	axisSlave:=             arrAxis[AxiseNo.VirAxisName.VirMain], 
	axisMaster:=          arrAxis[AxiseNo.VirAxisName.VirDriver]    , 
	bCreatTableDone=> , 
	bCreatTableError=> , 
	bError=>  );

fbCreatCamVirGMDriver.bCreatTableDone;
fbCreatCamVirGMDriver.bCreatTableError;
fbCreatCamVirGMDriver.bError;

(***********隔膜摆臂凸轮表**************)
fbCreatCamGMDanserMove(
	bCreatTable:=                     fbCreatCamGMDanserMove.bCreatTable, 
	Reset:=                                stSysState.bReset  , 
	iTable_L:=                            TableNo.M_GMDanserMove_L , //3
	iTable_R:=                           TableNo.M_GMDanserMove_R, //6
    fMoveLength:=                     fMaxPos-fMinPos , 
    fMasterKeyPos:=                   250  , //180
	axisSlave:=                           arrAxis[AxiseNo.VirAxisName.VirMain]  , 
	axisMaster:=                        arrAxis[AxiseNo.AxisName.SEPTATLine] , 
	bCreatTableDone=> , 
	bCreatTableError=> , 
	bError=>  );

fbCreatCamGMDanserMove.bCreatTableDone;
fbCreatCamGMDanserMove.bCreatTableError;
fbCreatCamGMDanserMove.bError;


(***********************************************************隔膜缓存凸轮表创建V2***20240229**************************************************************************)
(*******极片缓存电机*********)
fbCreatCamGMBuffer2_L(
	Reset:=                              stSysState.bReset  , 
	bCreatTable:=                   fbCreatCamGMBuffer2_L.bCreatTable, 
	iTable:=                            TableNo.M_GMBuffer2_L , 
	iTableGMVirDriver:=          TableNo.M_GMWind2_L  , 
	iTableGMStackCalculate:=  TableNo.M_GMLengthCalculate2_L , 
	iTableGMStackMove:=       TableNo.M_GMDanserMove_L , 
	fMaxPos:=                           fMaxPos, 
	fMinPos:=                            fMinPos , 
    iCcwSel :=                          1 , 
	arrGMCalculateTableData:= arrDeltaGMLength2_L , 

	axisSlave:=                     arrAxis[AxiseNo.AxisName.SEPTATCache], 
	axisMaster:=                  arrAxis[AxiseNo.VirAxisName.VirMain] , 
	bCreatTableDone=> , 
	bCreatTableError=> , 
	bError=>  );
fbCreatCamGMBuffer2_L.bCreatTableDone;
fbCreatCamGMBuffer2_L.bCreatTableError;
fbCreatCamGMBuffer2_L.bError;


(*******极片缓存电机*********)
fbCreatCamGMBuffer2_R(
	Reset:=                              stSysState.bReset  , 
	bCreatTable:=                    fbCreatCamGMBuffer2_R.bCreatTable, 
	iTable:=                             TableNo.M_GMBuffer2_R , 
	iTableGMVirDriver:=           TableNo.M_GMWind2_R  , 
	iTableGMStackCalculate:=   TableNo.M_GMLengthCalculate2_R , 
	iTableGMStackMove:=         TableNo.M_GMDanserMove_R , 
    iCcwSel :=                           2 , 
   	fMaxPos:=                           fMaxPos, 
	fMinPos:=                            fMinPos , 
	arrGMCalculateTableData:= arrDeltaGMLength2_R , 

	axisSlave:=                     arrAxis[AxiseNo.AxisName.SEPTATCache], 
	axisMaster:=                  arrAxis[AxiseNo.VirAxisName.VirMain] , 
	bCreatTableDone=> , 
	bCreatTableError=> , 
	bError=>  );
fbCreatCamGMBuffer2_R.bCreatTableDone;
fbCreatCamGMBuffer2_R.bCreatTableError;
fbCreatCamGMBuffer2_R.bError;


(***********隔膜放卷虚轴*凸轮表**************)
fbCreatCamVirGMDriver2(
	bCreatTable:=         fbCreatCamVirGMDriver2.bCreatTable , 
	Reset:=                  stSysState.bReset, 
	iTable_L:=               TableNo.M_GMWind2_L , 
	iTable_R:=               TableNo.M_GMWind2_R , 

	fGMLength_L:=		arrDeltaGMLength2_L[3600,1], 
	fGMLength_R:=	arrDeltaGMLength2_R[3600,1],  

	axisSlave:=            arrAxis[AxiseNo.VirAxisName.VirDriver], 
	axisMaster:=        arrAxis[AxiseNo.VirAxisName.VirMain]       , 
	bCreatTableDone=> , 
	bCreatTableError=> , 
	bError=>  );

fbCreatCamVirGMDriver2.bCreatTableDone;
fbCreatCamVirGMDriver2.bCreatTableError;
fbCreatCamVirGMDriver2.bError;


tGMCreateCamTON(IN:= , PT:=T#0.5S , Q=> , ET=> );
IF Mach_Control.U.DT_iMode=3 OR Mach_Control.U.DT_iMode=0 THEN//在手动状态下
			//从触据屏创建隔膜缓存凸轮
			rGMCreateCam_TRIG(CLK:=Mach_Control.DT_b.CreateCamStart2 , Q=> );
			IF rGMCreateCam_TRIG.Q THEN
				tGMCreateCamTON.IN:=FALSE;
				GMCreatCamStep0:=10;
				Mach_Control.DT_b.Error[1]:=FALSE;
			END_IF
END_IF			
			//隔膜缓存凸轮创建 
			CASE GMCreatCamStep0 OF
						10:
								IF NOT 	tGMCreateCamTON.Q THEN
										fbCreatCamVirGMDriver.bCreatTable:=FALSE;//放卷凸轮创建
										fbCreatCamGMDanserMove.bCreatTable:=FALSE;//	隔膜平移凸轮创建
										fbCreatCamGMBuffer_L.bCreatTable:=FALSE;//缓存左凸轮生成
										fbCreatCamGMBuffer_R.bCreatTable:=FALSE;//缓存右轮生成
										Mach_Control.DT_b.CreateCamDone2:=FALSE;
										tGMCreateCamTON.IN:=TRUE;
								ELSE
										tGMCreateCamTON.IN:=FALSE;
										GMCreatCamStep0:=11;
								END_IF
			
						11:
							IF  NOT DT_Cam_ton[3].Q THEN
								arrAxisCtrl[AxiseNo.AxisName.SEPTAunwinding].Cmd.bStop:=TRUE;
								arrAxisCtrl[AxiseNo.AxisName.SEPTATCache].Cmd.bStop:=TRUE;
								arrAxisCtrl[AxiseNo.AxisName.SEPTATLine].Cmd.bStop:=TRUE;
								DT_Cam_ton[3].IN:=TRUE;
							ELSE
								DT_Cam_ton[3].IN:=FALSE;
								GMCreatCamStep0:=12;
								arrAxisCtrl[AxiseNo.AxisName.SEPTAunwinding].Cmd.bStop:=FALSE;
								arrAxisCtrl[AxiseNo.AxisName.SEPTATCache].Cmd.bStop:=FALSE;
								arrAxisCtrl[AxiseNo.AxisName.SEPTATLine].Cmd.bStop:=FALSE;
							END_IF
					
						12:
							IF  NOT DT_Cam_ton[4].Q THEN
								arrAxisCtrl[AxiseNo.AxisName.SEPTAunwinding].Cmd.bReset:=TRUE;	
								arrAxisCtrl[AxiseNo.AxisName.SEPTATCache].Cmd.bReset:=TRUE;
								arrAxisCtrl[AxiseNo.AxisName.SEPTATLine].Cmd.bReset:=TRUE;		
								DT_Cam_ton[4].IN:=TRUE;
							 ELSE
								 DT_Cam_ton[4].IN:=FALSE;
								 GMCreatCamStep0:=13;
								arrAxisCtrl[AxiseNo.AxisName.SEPTAunwinding].Cmd.bReset:=FALSE;	
								arrAxisCtrl[AxiseNo.AxisName.SEPTATCache].Cmd.bReset:=FALSE;
								arrAxisCtrl[AxiseNo.AxisName.SEPTATLine].Cmd.bReset:=FALSE;		
							 END_IF
								
						13:
							arrAxisCtrl[AxiseNo.AxisName.SEPTAunwinding].Cmd.bEnable:=TRUE;
							arrAxisCtrl[AxiseNo.AxisName.SEPTATCache].Cmd.bEnable:=TRUE;
							arrAxisCtrl[AxiseNo.AxisName.SEPTATLine].Cmd.bEnable:=TRUE;
							IF arrAxisCtrl[AxiseNo.AxisName.SEPTAunwinding].Status.Enabled AND arrAxisCtrl[AxiseNo.AxisName.SEPTATCache].Status.Enabled AND
								arrAxisCtrl[AxiseNo.AxisName.SEPTATLine].Status.Enabled THEN
								 GMCreatCamStep0:=20;
							END_IF				
								
							
						20://隔膜变化长度度算
								iSetp1:=10;
								iSetp2:=10;
								Mach_Control.DT_b.CreateCamDone2:=FALSE;
								GMCreatCamStep0:=30;
						30://等待隔膜变化长度计算完成
								IF iSetp1=666 AND iSetp2=666 THEN
									GMCreatCamStep0:=40;
								END_IF
						40://创建放卷凸轮、隔膜平移凸轮
								fbCreatCamVirGMDriver.bCreatTable:=TRUE;//放卷凸轮创建
								 fbCreatCamGMDanserMove.bCreatTable:=TRUE;//	隔膜平移凸轮创建
								 fbCreatCamVirGMDriver2.bCreatTable:=TRUE;//放卷凸轮创建
								 
								GMCreatCamStep0:=50;	
						50://等待凸轮创建完成
								IF fbCreatCamVirGMDriver.bCreatTableDone AND fbCreatCamGMDanserMove.bCreatTableDone AND  fbCreatCamVirGMDriver2.bCreatTableDone  THEN
									GMCreatCamStep0:=60;	
								ELSE
										IF fbCreatCamVirGMDriver.bCreatTableError OR fbCreatCamGMDanserMove.bCreatTableError OR   fbCreatCamVirGMDriver2.bCreatTableError  THEN
												Mach_Control.DT_b.Error[1]:=TRUE;//隔膜缓存凸轮创建失败
												GMCreatCamStep0:=9999;		
										END_IF					
								END_IF
						60://创建隔膜缓存凸轮
							fbCreatCamGMBuffer_L.bCreatTable:=TRUE;//缓存左凸轮生成
							fbCreatCamGMBuffer_R.bCreatTable:=TRUE;//缓存右轮生成
							fbCreatCamGMBuffer2_L.bCreatTable:=TRUE;//缓存左凸轮生成
							fbCreatCamGMBuffer2_R.bCreatTable:=TRUE;//缓存右轮生成		
							
							 //fbCamInVirGM.bCreatTable:=TRUE;//隔膜虚轴凸轮生成
							GMCreatCamStep0:=70;	
						70://等待凸轮创建完成
							IF fbCreatCamGMBuffer_L.bCreatTableDone AND fbCreatCamGMBuffer_R.bCreatTableDone (*  AND fbCamInVirGM.bCreatTableDone *)    AND 
                                fbCreatCamGMBuffer2_L.bCreatTableDone AND  fbCreatCamGMBuffer2_R.bCreatTableDone THEN
								Mach_Control.DT_b.CreateCamDone2:=TRUE;//隔膜缓存凸轮创建完成
								GMCreatCamStep0:=6666;	
							ELSE
									IF fbCreatCamGMBuffer_L.bCreatTableError OR fbCreatCamGMBuffer_R.bCreatTableError  OR 
                                         fbCreatCamGMBuffer2_L.bCreatTableError AND  fbCreatCamGMBuffer2_R.bCreatTableError THEN
										Mach_Control.DT_b.Error[1]:=TRUE;//隔膜缓存凸轮创建失败
										GMCreatCamStep0:=9999;	
									END_IF
							END_IF
			END_CASE
(************************************************************凸轮耦合*****************************************************************************)
//隔膜放卷凸轮
fbCamInVirGMDriver(  
	Reset:=                      stSysState.bReset  , 
	bCamInExecute:=       fbCamInVirGMDriver.bCamInExecute, 
	iTable1:=                   TableNo.M_GMWind_L  , //从左到右，正极到负极
	iTable2:=                  TableNo.M_GMWind_R  , //从右到左，负极到正极
	iTableSel:=                fbCamInVirGMDriver.iTableSel , //凸轮表号选择
	ParCamIn:= , 
 	axisMaster:=            arrAxis[AxiseNo.VirAxisName.VirMain], 
	axisSlave:=               arrAxis[AxiseNo.VirAxisName.VirDriver]    , 
	bError=> , 
	bReady=> , 
	bInSync=> );

Mach_Control.DT_b.Error[16]:=fbCamInVirGMDriver.bError;
fbCamInVirGMDriver.bReady;
fbCamInVirGMDriver.bInSync;


//隔膜平移凸轮
IF  fbCamInGMDanserMove.iTableSel=2 THEN
     fbCamInGMDanserMove.ParCamIn.SlaveOffset:=-(fMaxPos-fMinPos);
ELSE
    fbCamInGMDanserMove.ParCamIn.SlaveOffset:=0;
END_IF

fbCamInGMDanserMove(
	Reset:=                      stSysState.bReset  , 
	bCamInExecute:=       fbCamInGMDanserMove.bCamInExecute, 
	iTable1:=                   TableNo.M_GMDanserMove_L  , 
	iTable2:=                   TableNo.M_GMDanserMove_R  , 
	iTableSel:=                fbCamInGMDanserMove.iTableSel , 
	ParCamIn:= , 
  	axisMaster:=            arrAxis[AxiseNo.VirAxisName.VirMain] , //VirMain
	axisSlave:=               arrAxis[AxiseNo.AxisName.SEPTATLine] , 
	bError=> , 
	bReady=> , 
	bInSync=> );

Mach_Control.DT_b.Error[17]:=fbCamInGMDanserMove.bError;
fbCamInGMDanserMove.bReady;
fbCamInGMDanserMove.bInSync;

//隔膜缓存凸轮
fbCamInGMBuffer.ParCamIn.MasterScaling:=0.1;
fbCamInGMBuffer(
	Reset:=                      stSysState.bReset  , 
	bCamInExecute:=       fbCamInGMBuffer.bCamInExecute, 
	iTable1:=                   TableNo.M_GMBuffer_L  , 
	iTable2:=                   TableNo.M_GMBuffer_R  , 
	iTableSel:=                fbCamInGMBuffer.iTableSel , 
	ParCamIn:= , 
  	axisMaster:=           arrAxis[AxiseNo.VirAxisName.VirMain] , 
	axisSlave:=               arrAxis[AxiseNo.AxisName.SEPTATCache] , 
	bError=> , 
	bReady=> , 
	bInSync=> );

Mach_Control.DT_b.Error[18]:=fbCamInGMBuffer.bError;
fbCamInGMBuffer.bReady;
fbCamInGMBuffer.bInSync;



(************************************************************凸轮耦合V2*****************************************************************************)
//隔膜放卷凸轮
fbCamInVirGMDriver2(  
	Reset:=                      stSysState.bReset  , 
	bCamInExecute:=       fbCamInVirGMDriver2.bCamInExecute, 
	iTable1:=                   TableNo.M_GMWind2_L  , //从左到右，正极到负极
	iTable2:=                  TableNo.M_GMWind2_R  , //从右到左，负极到正极
	iTableSel:=                fbCamInVirGMDriver2.iTableSel , //凸轮表号选择
	ParCamIn:= , 
 	axisMaster:=            arrAxis[AxiseNo.VirAxisName.VirMain], 
	axisSlave:=               arrAxis[AxiseNo.VirAxisName.VirDriver]    , 
	bError=> , 
	bReady=> , 
	bInSync=> );

fbCamInVirGMDriver2.bError;
fbCamInVirGMDriver2.bReady;
fbCamInVirGMDriver2.bInSync;


//隔膜缓存凸轮
fbCamInGMBuffer2.ParCamIn.MasterScaling:=0.1;
fbCamInGMBuffer2(
	Reset:=                      stSysState.bReset  , 
	bCamInExecute:=       fbCamInGMBuffer2.bCamInExecute, 
	iTable1:=                   TableNo.M_GMBuffer2_L  , 
	iTable2:=                   TableNo.M_GMBuffer2_R  , 
	iTableSel:=                fbCamInGMBuffer2.iTableSel , 
	ParCamIn:= , 
  	axisMaster:=           arrAxis[AxiseNo.VirAxisName.VirMain] , 
	axisSlave:=               arrAxis[AxiseNo.AxisName.SEPTATCache] , 
	bError=> , 
	bReady=> , 
	bInSync=> );

fbCamInGMBuffer2.bError;
fbCamInGMBuffer2.bReady;
fbCamInGMBuffer2.bInSync;












(*

(***********************************************************隔膜缓存凸轮表创建*****************************************************************************)
(*******极片缓存电机*********)
fbCreatCamGMBuffer_L.iKeyPosTemp:=20;
fbCreatCamGMBuffer_L(
	Reset:=                              stSysState.bReset  , 
	bCreatTable:=                   fbCreatCamGMBuffer_L.bCreatTable, 
	iTable:=                            TableNo.M_GMBuffer_L , //10
	iTableGMVirDriver:=          TableNo.M_GMWind_L  , //1
	iTableGMStackCalculate:=  TableNo.M_GMLengthCalculate_L , //2
	iTableGMStackMove:=       TableNo.M_GMDanserMove_L , //3
	fMaxPos:=                           fMaxPos, 
	fMinPos:=                            fMinPos , 
    iCcwSel :=                          1 , 
	arrGMCalculateTableData:= arrDeltaGMLength_L , 

	axisSlave:=                     arrAxis[AxiseNo.VirAxisName.VirMain], 
	axisMaster:=                  arrAxis[AxiseNo.AxisName.SEPTATCache] , 
	bCreatTableDone=> , 
	bCreatTableError=> , 
	bError=>  );
fbCreatCamGMBuffer_L.bCreatTableDone;
fbCreatCamGMBuffer_L.bCreatTableError;
fbCreatCamGMBuffer_L.bError;


(*******极片缓存电机*********)
fbCreatCamGMBuffer_R.iKeyPosTemp:=20;
fbCreatCamGMBuffer_R(
	Reset:=                              stSysState.bReset  , 
	bCreatTable:=                    fbCreatCamGMBuffer_R.bCreatTable, 
	iTable:=                             TableNo.M_GMBuffer_R , //20
	iTableGMVirDriver:=           TableNo.M_GMWind_R  , //4
	iTableGMStackCalculate:=   TableNo.M_GMLengthCalculate_R , //5
	iTableGMStackMove:=         TableNo.M_GMDanserMove_R , //6
    iCcwSel :=                           2 , //2
   	fMaxPos:=                           fMaxPos, 
	fMinPos:=                            fMinPos , 
	arrGMCalculateTableData:= arrDeltaGMLength_R , 

	axisSlave:=                     arrAxis[AxiseNo.VirAxisName.VirMain], 
	axisMaster:=                  arrAxis[AxiseNo.AxisName.SEPTATCache] , 
	bCreatTableDone=> , 
	bCreatTableError=> , 
	bError=>  );
fbCreatCamGMBuffer_R.bCreatTableDone;
fbCreatCamGMBuffer_R.bCreatTableError;
fbCreatCamGMBuffer_R.bError;


(***********隔膜放卷虚轴*凸轮表**************)
fbCreatCamVirGMDriver(
	bCreatTable:=         fbCreatCamVirGMDriver.bCreatTable , 
	Reset:=                  stSysState.bReset, 
	iTable_L:=               TableNo.M_GMWind_L , //1
	iTable_R:=               TableNo.M_GMWind_R , //4

	fGMLength_L:=       arrDeltaGMLength_L[3600,1]+1.2 , 
	fGMLength_R:=       arrDeltaGMLength_R[3600,1]+1.2 , 

	axisSlave:=             arrAxis[AxiseNo.VirAxisName.VirMain], 
	axisMaster:=          arrAxis[AxiseNo.VirAxisName.VirDriver]    , 
	bCreatTableDone=> , 
	bCreatTableError=> , 
	bError=>  );

fbCreatCamVirGMDriver.bCreatTableDone;
fbCreatCamVirGMDriver.bCreatTableError;
fbCreatCamVirGMDriver.bError;
*)
END_ACTION

ACTION GMBufferLengthCalculate:
(**************************************************************************隔膜计算V2******************************************)


(**************************************************************************隔膜变化长度计算********************************************)
//隔膜垂直向下为隔膜摆臂的机械零点
//C1点坐标=当前坐标+隔膜辊半径
//fMaxPos=隔膜摆臂右目标位置+隔膜辊半径

(*
//C1活动范围   -188.05------164.05        从右到左 
(**********坐标自动计算**********)
Par.Mechaical.fGMRollDiameter:=24;
IF Par.Mechaical.fGM_X>0 AND Par.Mechaical.fGM_Y>0 THEN
	Par.Mechaical.y_B1:=Par.Mechaical.fGM_Y-Par.Mechaical.fGMRollDiameter/2;
	Par.Mechaical.y_C1:=Par.Mechaical.y_B1-72;
	//Par.Mechaical.y_A5:=Par.Mechaical.y_B1+333;
	Par.Mechaical.x_D2:=Par.Mechaical.fGM_X+52.5;
	Par.Mechaical.x_D1:=Par.Mechaical.x_D2-par.stDT_date.Width;
END_IF
IF Par.Mechaical.fGM_Z>0 THEN
	Par.Mechaical.y_A5:=Par.Mechaical.fGM_Z+Par.Mechaical.fGMRollDiameter/2;
END_IF
*)
       
arrAxisPar [AxiseNo.AxisName.SEPTATLine].arrTargetPoint[1];//左
arrAxisPar [AxiseNo.AxisName.SEPTATLine].arrTargetPoint[2];//右
Par.Mechaical.fGMRollDiameter;
CASE  iSetp1  OF   
10://计算相间距
    I10:=0;
	//fMaxPos:=arrAxisPar [AxiseNo.AxisName.SEPTATLine].arrTargetPoint[2]-arrAxisPar [AxiseNo.AxisName.SEPTATLine].arrTargetPoint[3] -Par.Mechaical.fGMRollDiameter/2;
	//fMinPos:=arrAxisPar [AxiseNo.AxisName.SEPTATLine].arrTargetPoint[1]-arrAxisPar [AxiseNo.AxisName.SEPTATLine].arrTargetPoint[3] -Par.Mechaical.fGMRollDiameter/2;	
	fMaxPos:=arrAxisPar [AxiseNo.AxisName.SEPTATLine].arrTargetPoint[2]-Par.Mechaical.fGMRollDiameter/2;
	fMinPos:=arrAxisPar [AxiseNo.AxisName.SEPTATLine].arrTargetPoint[1]-Par.Mechaical.fGMRollDiameter/2;
  // fMaxPos:=164.05;         //  =隔膜摆臂当前位置-r              隔膜摆臂中间为0位置
   //fMinPos:=-200;          //  =隔膜摆臂当前位置-r              隔膜摆臂中间为0位置          -188.55
    iNumberOfPoint:=3600;
    fInterval:=(fMaxPos-fMinPos)/ iNumberOfPoint ;


    fradii:= Par.Mechaical.fGMRollDiameter/2 ;
    fJumpPos:=-fradii;
    k_Comp:=fcompensationPos/(fMaxPos-fJumpPos) ;
	bMoveFowerdR:=FALSE;
    iSetp1:=20;

20:
   fTagatPos:=fMaxPos-I10*fInterval;
   bExecute:=TRUE;
   bExecute2:=TRUE;
    iSetp1:=30;
30:
   IF NOT  bExecute   AND  NOT bExecute2   THEN
        arrfTagatPos_R[I10]:=fTagatPos;
        arrDeltaGMLength_R[I10,0]:=I10;
 
       arrGMLengthDown_R[I10] :=fbGMLengthV1_R.fTotalLenght;
       arrGMLengthUp_R[I10] :=fbGMLengthV2_R.fTotalLenght   ;
		
       arrDeltaGMLength_R[0,1]:=0;
       IF I10>=1 THEN
         arrDeltaGMLength_R[I10,1]:=arrGMLengthDown_R[I10]+arrGMLengthUp_R[I10]-(arrGMLengthDown_R[0]+arrGMLengthUp_R[0] )        ;
      END_IF
          I10:=I10+1;
		IF I10>iNumberOfPoint THEN
			iSetp1:=100;  
		ELSE
			iSetp1:=20;  
		 END_IF
   END_IF

100:
       I10:=0;
	//fMaxPos:=arrAxisPar [AxiseNo.AxisName.SEPTATLine].arrTargetPoint[2]-arrAxisPar [AxiseNo.AxisName.SEPTATLine].arrTargetPoint[3] -Par.Mechaical.fGMRollDiameter/2;
	//fMinPos:=arrAxisPar [AxiseNo.AxisName.SEPTATLine].arrTargetPoint[1]-arrAxisPar [AxiseNo.AxisName.SEPTATLine].arrTargetPoint[3] -Par.Mechaical.fGMRollDiameter/2;	
	fMaxPos:=arrAxisPar [AxiseNo.AxisName.SEPTATLine].arrTargetPoint[2]-Par.Mechaical.fGMRollDiameter/2;
	fMinPos:=arrAxisPar [AxiseNo.AxisName.SEPTATLine].arrTargetPoint[1]-Par.Mechaical.fGMRollDiameter/2;
  // fMaxPos:=164.05;         //  =隔膜摆臂当前位置-r              隔膜摆臂中间为0位置
   //fMinPos:=-200;          //  =隔膜摆臂当前位置-r              隔膜摆臂中间为0位置          -188.55
    iNumberOfPoint:=3600;
    fInterval:=(fMaxPos-fMinPos)/ iNumberOfPoint ;


    fradii:= Par.Mechaical.fGMRollDiameter/2 ;
    fJumpPos:=-fradii;
    k_Comp:=fcompensationPos/(fMaxPos-fJumpPos) ;
   bMoveFowerdR:=TRUE;
    iSetp1:=120;

120:
     fTagatPos:=fMaxPos-I10*fInterval;
     bExecute:=TRUE;
     bExecute2:=TRUE;
      iSetp1:=130;

130:
	IF NOT  bExecute   AND  NOT bExecute2   THEN
			arrfTagatPos2_R[I10]:=fTagatPos;
			arrDeltaGMLength2_R[I10,0]:=I10;
			
			arrGMLengthDown2_R[I10] :=fbGMLengthV1_R.fTotalLenght;
			arrDeltaGMLength2_R[0,1]:=0;
			IF I10>=1 THEN
				arrDeltaGMLength2_R[I10,1]:=arrGMLengthDown2_R[I10]+arrGMLengthUp_R[I10]-(arrGMLengthDown2_R[0]+arrGMLengthUp_R[0] )        ;
			END_IF
			I10:=I10+1;
			IF I10>iNumberOfPoint THEN
				iSetp1:=666;  
			ELSE
				iSetp1:=120;  
			END_IF
		END_IF 
END_CASE



//C1活动范围   -188.05------164.05        从左到右   
CASE  iSetp2  OF   
10://计算相间距
    I12:=0;
	fMaxPos:=arrAxisPar [AxiseNo.AxisName.SEPTATLine].arrTargetPoint[2]-Par.Mechaical.fGMRollDiameter/2;
	fMinPos:=arrAxisPar [AxiseNo.AxisName.SEPTATLine].arrTargetPoint[1]-Par.Mechaical.fGMRollDiameter/2;
  // fMaxPos:=164.05;       
   // fMinPos:=-200;  
    iNumberOfPoint:=3600;
    fInterval2:=(fMaxPos-fMinPos)/ iNumberOfPoint ;
 
    fradii:= Par.Mechaical.fGMRollDiameter/2 ;
    fJumpPos:=-fradii;
    k_Comp:=fcompensationPos/(fMaxPos-fJumpPos) ;

     arrDeltaGMLengthAbs_L[0,0]:=0 ;
	 bMoveFowerdL:=FALSE;
    iSetp2:=20;

20:
   fTagatPos2:=fMinPos+I12*fInterval2;
   bExecute3:=TRUE;
   bExecute4:=TRUE;
    iSetp2:=30;

30:
   IF NOT  bExecute3   AND  NOT bExecute4   THEN
        arrfTagatPos_L[I12]:=fTagatPos2;
        arrDeltaGMLength_L[I12,0]:=I12;
        arrDeltaGMLengthAbs_L[I12,0]:=fTagatPos2-fMinPos ;

        arrGMLengthDown_L[I12] :=  fbGMLengthV1_L.fTotalLenght;  //下
         arrGMLengthUp_L[I12] :=fbGMLengthV2_L.fTotalLenght   ;  //上	
		
      arrDeltaGMLength_L[0,1]:=0;
       IF I12>=1 THEN
         arrDeltaGMLength_L[I12,1]:=arrDeltaGMLengthAbs_L[I12,1]:= arrGMLengthDown_L[I12]+arrGMLengthUp_L[I12]-(arrGMLengthDown_L[0]+arrGMLengthUp_L[0] )   ;
      END_IF
          I12:=I12+1;
		IF I12>iNumberOfPoint THEN
			iSetp2:=100;  
		ELSE
			iSetp2:=20;  
		 END_IF
   END_IF

100:
    I12:=0;
	fMaxPos:=arrAxisPar [AxiseNo.AxisName.SEPTATLine].arrTargetPoint[2]-Par.Mechaical.fGMRollDiameter/2;
	fMinPos:=arrAxisPar [AxiseNo.AxisName.SEPTATLine].arrTargetPoint[1]-Par.Mechaical.fGMRollDiameter/2;
  // fMaxPos:=164.05;       
   // fMinPos:=-200;  
    iNumberOfPoint:=3600;
    fInterval2:=(fMaxPos-fMinPos)/ iNumberOfPoint ;
 
    fradii:= Par.Mechaical.fGMRollDiameter/2 ;
    fJumpPos:=-fradii;
    k_Comp:=fcompensationPos/(fMaxPos-fJumpPos) ;

     arrDeltaGMLength2Abs_L[0,0]:=0 ;
	 bMoveFowerdL:=TRUE;
    iSetp2:=120;
	 
120:	 
	   fTagatPos2:=fMinPos+I12*fInterval2;
	   bExecute3:=TRUE;
	   bExecute4:=TRUE;
		iSetp2:=130;	 
130:	 
  IF NOT  bExecute3   AND  NOT bExecute4   THEN
        arrfTagatPos2_L[I12]:=fTagatPos2;
        arrDeltaGMLength2_L[I12,0]:=I12;
        arrDeltaGMLength2Abs_L[I12,0]:=fTagatPos2-fMinPos ;
		
        arrGMLengthDown2_L[I12] :=  fbGMLengthV1_L.fTotalLenght;  //下
       // arrGMLengthUp_L[I12] :=fbGMLengthV2_L.fTotalLenght   ;  //上	
      arrDeltaGMLength2_L[0,1]:=0;
       IF I12>=1 THEN
         arrDeltaGMLength2_L[I12,1]:=arrDeltaGMLength2Abs_L[I12,1]:= arrGMLengthDown2_L[I12]+arrGMLengthUp_L[I12]-(arrGMLengthDown2_L[0]+arrGMLengthUp_L[0] )  ;
      END_IF
          I12:=I12+1;
		IF I12>iNumberOfPoint THEN
			iSetp2:=666;  
		ELSE
			iSetp2:=120;  
		 END_IF

   END_IF	 
	
END_CASE


(***从右往左运动*)
fbGMLengthV1_R(
	bExecute:=           bExecute , 
     x_C1:=                  fTagatPos, 

    fradii:=                       Par.Mechaical.fGMRollDiameter/2 , 
    y_C1:=                       Par.Mechaical.y_C1    , 
    x_D1:=                      SEL(bMoveFowerdR,Par.Mechaical.x_D1,Par.Mechaical.x_D1)    , //
    x_D2:=                      SEL(bMoveFowerdR,Par.Mechaical.x_D2,Par.Mechaical.x_D1)  , //20221028  SJ
	fDegree=> , 
	fArcLength=> , 
	fLineLength=> , 
	fTotalLenght=> );
fbGMLengthV1_R.fArcLength;
fbGMLengthV1_R.fDegree;
fbGMLengthV1_R.fLineLength;
fbGMLengthV1_R.fTotalLenght;


(*
fbGMLengthV2_R(
	x_C1:=                           fTagatPos , 

   fradii:=                       Par.Mechaical.fGMRollDiameter/2 , 
    y_C1:=                       Par.Mechaical.y_C1    , 
    x_D1:=                       Par.Mechaical.x_D1   , 
    x_D2:=                       Par.Mechaical.x_D2  , 
    y_B1:=                       Par.Mechaical.y_B1   , 
    y_A5:=                       Par.Mechaical.y_A5   , 

	fDegree=> , 
	fArcLength=> , 
	fLineLength=> , 
	fTotalLenght=> , 
	bExecute:=                    bExecute2 );

fbGMLengthV2_R.fArcLength;
fbGMLengthV2_R.fDegree;
fbGMLengthV2_R.fLineLength;
fbGMLengthV2_R.fTotalLenght;
*)

fbGMLengthV2_R(
	x_C1:=                           fTagatPos , 

   fradii:=                       Par.Mechaical.fGMRollDiameter/2 , 
    y_C1:=                       Par.Mechaical.y_C1    , 
    x_D1:=                       Par.Mechaical.x_D1   , 
    x_D2:=                       Par.Mechaical.x_D2  , 
    y_B1:=                       Par.Mechaical.y_B1   , 
    y_A5:=                       Par.Mechaical.y_A5   , 

	fDegree=> , 
	fArcLength=> , 
	fLineLength=> , 
	fTotalLenght=> , 
	bExecute:=                    bExecute2 );

fbGMLengthV2_R.fArcLength;
fbGMLengthV2_R.fDegree;
fbGMLengthV2_R.fLineLength;
fbGMLengthV2_R.fTotalLenght;


(***从左往右运动*)
fbGMLengthV1_L(  //下
	bExecute:=             bExecute3 , 
     x_C1:=                  fTagatPos2, 

    fradii:=                       Par.Mechaical.fGMRollDiameter/2 , 
    y_C1:=                       Par.Mechaical.y_C1    , 
    x_D1:=                         SEL(bMoveFowerdL,Par.Mechaical.x_D1,Par.Mechaical.x_D2)  , // x_D1:=x_D2;//20221028SJ
    x_D2:=                       SEL(bMoveFowerdL,Par.Mechaical.x_D2,Par.Mechaical.x_D2)  , // x_D1:=x_D2;//20221028SJ

	fDegree=> , 
	fArcLength=> , 
	fLineLength=> , 
	fTotalLenght=> );
fbGMLengthV1_L.fArcLength;
fbGMLengthV1_L.fDegree;
fbGMLengthV1_L.fLineLength;
fbGMLengthV1_L.fTotalLenght;


(*
fbGMLengthV2_L( //上
	x_C1:=                        fTagatPos2 , 
    
    fradii:=                       Par.Mechaical.fGMRollDiameter/2 , 
    y_C1:=                       Par.Mechaical.y_C1    , 
    x_D1:=                       Par.Mechaical.x_D1   , 
    x_D2:=                       Par.Mechaical.x_D2  , 
    y_B1:=                       Par.Mechaical.y_B1   , 
    y_A5:=                       Par.Mechaical.y_A5   , 

	fDegree=> , 
	fArcLength=> , 
	fLineLength=> , 
	fTotalLenght=> , 
	bExecute:=                    bExecute4 );

fbGMLengthV2_L.fArcLength;
fbGMLengthV2_L.fDegree;
fbGMLengthV2_L.fLineLength;
fbGMLengthV2_L.fTotalLenght;
*)
fbGMLengthV2_L( //上
	x_C1:=                        fTagatPos2 , 
    
    fradii:=                       Par.Mechaical.fGMRollDiameter/2 , 
    y_C1:=                       Par.Mechaical.y_C1    , 
    x_D1:=                       Par.Mechaical.x_D1   , 
    x_D2:=                       Par.Mechaical.x_D2  , 
    y_B1:=                       Par.Mechaical.y_B1   , 
    y_A5:=                       Par.Mechaical.y_A5   , 

	fDegree=> , 
	fArcLength=> , 
	fLineLength=> , 
	fTotalLenght=> , 
	bExecute:=                    bExecute4 );

fbGMLengthV2_L.fArcLength;
fbGMLengthV2_L.fDegree;
fbGMLengthV2_L.fLineLength;
fbGMLengthV2_L.fTotalLenght;




fbReadCamSlavePos(
	Execute:=              fbReadCamSlavePos.Execute , 
	CamTableID:=        1, 
	MasterPosition:=    fbReadCamSlavePos.MasterPosition, 
	Done=> , 
	Busy=> , 
	Error=> , 
	ErrorID=> , 
	SlavePosition=> , 
	SlaveVelocity=> , 
	SlaveAcceleration=> );

fbReadCamSlavePos.Done;
fbReadCamSlavePos.Error;
fbReadCamSlavePos.SlavePosition;
END_ACTION

ACTION GMEmptyFold1:
//首层隔膜空叠自动步	iEmptyFoldStep[1]
DT_AlarmTon[5](IN:=  , PT:=T#300MS , Q=> , ET=> );
	
IF Mach_Control.U.DT_iMode=1 THEN//在自动状态下
CASE iEmptyFoldStep[1] OF
100:
   DT_AlarmTon[5].IN:=FALSE;
   IF NOT DP_SinStepe THEN
		IF NOT  Mach_Control.DT_b.DT_YDOpenwindow THEN
			CCD.Over.Start.iPliesNo:=UINT_TO_INT(Mach_Control.Ca_b.Ca_Quantited + Mach_Control.An_b.An_Quantited);
			CCD.Over.Finish.OverhandResult:=0;
			Mach_Control.DT_b.OverhandResult:=0;
			CCD.Over.Start.iPhotoDo:=3;
			Mach_Control.DT_b.CDD_OverStart:=TRUE;
			iEmptyFoldStep[1]:=200;
		ELSE
			iEmptyFoldStep[1]:=900;
		END_IF
    END_IF
200:
DT_AlarmTon[5].IN:=TRUE;
IF Mach_Control.DT_b.OverhandResult=1 THEN
	CellMemory[Mach_Control.DT_b.DT_Memory].Overhang_Result[CCD.Over.Start.iPliesNo]:=Mach_Control.DT_b.OverhandResult;
	iEmptyFoldStep[1]:=900;
ELSIF Mach_Control.DT_b.OverhandResult=5 THEN
	Mach_Control.DT_b.Error[63]:=TRUE;//首次对齐度拍照NG，请调节压刀间距
	iEmptyFoldStep[1]:=100;
ELSIF DT_AlarmTon[5].Q THEN
	Mach_Control.DT_b.Error[65]:=TRUE;//压刀间距测量结果返馈超时
	iEmptyFoldStep[1]:=100;
	DT_AlarmTon[5].IN :=FALSE;
END_IF



900://判断主轴是否停止、是否在初始位、是否有轴在耦合中
	bEmptyFoldMark[1]:=TRUE;//进入空叠流程
	IF NOT DP_SinStepe THEN
		bFirstFoldFinish[1]:=FALSE;//首层隔膜空叠完成
		IF arrAxisCtrl[AxiseNo.VirAxisName.VirMain].Status.NoMoving AND arrAxisCtrl[AxiseNo.VirAxisName.VirMain].Status.fSetPos=0 AND NOT DT_AxiseCoupling THEN
			DT_SingeMode();//单步选择	
			iEmptyFoldStep[1]:=1020;
		ELSE
			DT_SingeMode();//单步选择	
			DP_Step1:=100;//解除耦合，主轴回零
			iEmptyFoldStep[1]:=1010;
		END_IF
	END_IF
1010://判断主轴当前的当前位置是否为0
	IF DP_Step1=6666 AND arrAxisCtrl[AxiseNo.VirAxisName.VirMain].Status.NoMoving AND arrAxisCtrl[AxiseNo.VirAxisName.VirMain].Status.fSetPos=0 AND NOT DT_AxiseCoupling THEN
		DT_SingeMode();//单步选择
		iEmptyFoldStep[1]:=1020;						
	END_IF	

1020://判断NG气缸是否在安全位
	IF arrCyCtrl[arrCyNo.CylinderName.AnScrapbinCy].Status.ONState AND arrCyCtrl[arrCyNo.CylinderName.CaScrapbinUDCy].Status.OFFState AND
		arrCyCtrl[arrCyNo.CylinderName.CaScrapbinCy].Status.ONState AND arrCyCtrl[arrCyNo.CylinderName.PreDiaph].Status.OFFState AND 
		arrCyCtrl[arrCyNo.CylinderName.PoleHotCutterCy].Status.OFFState AND arrCyCtrl[arrCyNo.CylinderName.PoleTapeCy].Status.OFFState AND
		arrCyCtrl[arrCyNo.CylinderName.PoleTapeSplicerRCy].Status.ONState AND arrCyCtrl[arrCyNo.CylinderName.PoleTapeSplicerLCy].Status.ONState THEN
		iEmptyFoldStep[1]:=1050;		
	ELSE
		iEmptyFoldStep[1]:=1030;	
	END_IF
1030:
	IF NOT DP_SinStepe THEN
		arrCyCtrl[arrCyNo.CylinderName.AnScrapbinCy].Cmd.bON:=TRUE;
		arrCyCtrl[arrCyNo.CylinderName.PreDiaph].Cmd.bOFF:=TRUE;
		arrCyCtrl[arrCyNo.CylinderName.PoleHotCutterCy].Cmd.bOFF:=TRUE;
		arrCyCtrl[arrCyNo.CylinderName.PoleTapeCy].Cmd.bOFF:=TRUE;
		arrCyCtrl[arrCyNo.CylinderName.PoleTapeSplicerRCy].Cmd.bON:=TRUE;
		arrCyCtrl[arrCyNo.CylinderName.PoleTapeSplicerLCy].Cmd.bON:=TRUE;
		arrCyCtrl[arrCyNo.CylinderName.CaScrapbinCy].Cmd.bON:=TRUE;
		IF   arrCyCtrl[arrCyNo.CylinderName.AnScrapbinCy].Status.ONState AND  arrCyCtrl[arrCyNo.CylinderName.PreDiaph].Status.OFFState AND 
		arrCyCtrl[arrCyNo.CylinderName.PoleHotCutterCy].Status.OFFState AND arrCyCtrl[arrCyNo.CylinderName.PoleTapeCy].Status.OFFState AND
		arrCyCtrl[arrCyNo.CylinderName.PoleTapeSplicerRCy].Status.ONState AND arrCyCtrl[arrCyNo.CylinderName.PoleTapeSplicerLCy].Status.ONState
		AND arrCyCtrl[arrCyNo.CylinderName.CaScrapbinCy].Cmd.bON THEN
			DT_SingeMode();//单步选择	
			iEmptyFoldStep[1]:=1040;									
		END_IF
	END_IF	
1040:
	IF NOT DP_SinStepe THEN
		arrCyCtrl[arrCyNo.CylinderName.CaScrapbinUDCy].Cmd.bOFF:=TRUE;
		IF  arrCyCtrl[arrCyNo.CylinderName.CaScrapbinUDCy].Status.OFFState THEN
			DT_SingeMode();//单步选择	
			iEmptyFoldStep[1]:=1050;	
		END_IF		
	END_IF				
1050://	首层空叠隔膜
	IF Mach_Control.An_b.An_FirstFoldCnt<=Mach_Control.Ca_b.Ca_FirstFoldCnt THEN//先叠正极
		iEmptyFoldStep[1]:=1100;
	ELSIF Mach_Control.An_b.An_FirstFoldCnt>Mach_Control.Ca_b.Ca_FirstFoldCnt  THEN//先叠负极
		iEmptyFoldStep[1]:=1500;
	END_IF	
1100://判断叠台搬运机械手是否有片
	IF AN_CarryingPos1  THEN//正极搬运、叠片各轴在初始位	
		IF arrCyCtrl[arrCyNo.ElectValveName.AnDTCarryingVacuum].Io.DIOnSwitch AND  Mach_Control.An_b.An_DPCarryingFalg THEN//正极再取片位且叠台搬运有片,把当前片放到纠偏台
			iEmptyFoldStep[1]:=1150;
		ELSE
			iEmptyFoldStep[1]:=2000;	
		END_IF
	ELSE
		Mach_Control.DT_b.Error[8]:=TRUE;//叠正极片凸轮耦合时，正极片不在取片位
		//DP_Step0:=10001;
	END_IF	
	
1150://纠偏台回初始位
	//纠偏平台X1移动至初始位
	IF NOT DP_SinStepe THEN
		IF arrAxisCtrl[AxiseNo.AxisName.AndeviationX1].Status.Homed  AND arrAxisCtrl[AxiseNo.AxisName.AndeviationX1].Status.NoMoving AND NOT  arrAxisCtrl[AxiseNo.AxisName.AndeviationX1].Status.Error THEN
			IF arrAxisCtrl[AxiseNo.AxisName.AndeviationX1].Cmd.arrbRealPoint[1] THEN
				arrAxisCtrl[AxiseNo.AxisName.AndeviationX1].Cmd.iGoSetPos:=0;
			ELSE
				arrAxisCtrl[AxiseNo.AxisName.AndeviationX1].Cmd.iGoSetPos:=1;
			END_IF					
		END_IF
		//纠偏平台X2移动至初始位
		IF arrAxisCtrl[AxiseNo.AxisName.AndeviationX2].Status.Homed  AND arrAxisCtrl[AxiseNo.AxisName.AndeviationX2].Status.NoMoving AND NOT  arrAxisCtrl[AxiseNo.AxisName.AndeviationX2].Status.Error THEN
			IF arrAxisCtrl[AxiseNo.AxisName.AndeviationX2].Cmd.arrbRealPoint[1] THEN
				arrAxisCtrl[AxiseNo.AxisName.AndeviationX2].Cmd.iGoSetPos:=0;
			ELSE
				arrAxisCtrl[AxiseNo.AxisName.AndeviationX2].Cmd.iGoSetPos:=1;
			END_IF					
		END_IF
		//纠偏平台X2移动至初始位
		IF arrAxisCtrl[AxiseNo.AxisName.AndeviationY].Status.Homed  AND arrAxisCtrl[AxiseNo.AxisName.AndeviationY].Status.NoMoving AND NOT  arrAxisCtrl[AxiseNo.AxisName.AndeviationY].Status.Error THEN
			IF arrAxisCtrl[AxiseNo.AxisName.AndeviationY].Cmd.arrbRealPoint[1] THEN
				arrAxisCtrl[AxiseNo.AxisName.AndeviationY].Cmd.iGoSetPos:=0;
			ELSE
				arrAxisCtrl[AxiseNo.AxisName.AndeviationY].Cmd.iGoSetPos:=1;
			END_IF					
		END_IF
		IF arrAxisCtrl[AxiseNo.AxisName.AndeviationX1].Cmd.arrbRealPoint[1] AND arrAxisCtrl[AxiseNo.AxisName.AndeviationX2].Cmd.arrbRealPoint[1] AND arrAxisCtrl[AxiseNo.AxisName.AndeviationY].Cmd.arrbRealPoint[1] THEN
			DT_SingeMode();//单步选择	
			iEmptyFoldStep[1]:=1200;	
		END_IF	
	END_IF
1200:
	IF NOT DP_SinStepe THEN
		IF arrAxisCtrl[AxiseNo.AxisName.AnDTCarryingUpDown].Cmd.arrbRealPoint[2] THEN
			arrAxisCtrl[AxiseNo.AxisName.AnDTCarryingUpDown].Cmd.iGoSetPos:=0;
			/// 吸盘破真空    纠偏台开真空
			arrCyCtrl[arrCyNo.ElectValveName.AnDTCarryingVacuum].Cmd.bON:=TRUE;	//正极叠台搬运升降真空	真空
			arrCyCtrl[arrCyNo.ElectValveName.AnDTCarryingVacuum].Cmd.bOFF:=FALSE;	//正极叠台搬运升降真空破真空		
			//arrCyCtrl[arrCyNo.ElectValveName.AnDTCarryingVacuumBark].Cmd.bON:=TRUE;	//正极叠台搬运升降真空	真空
			//arrCyCtrl[arrCyNo.ElectValveName.AnDTCarryingVacuumBark].Cmd.bOFF:=FALSE;	//正极叠台搬运升降真空破真空											
			arrCyCtrl[arrCyNo.ElectValveName.AndeviationVacuum].Cmd.bON:=TRUE;	//正极纠偏台真空			
			arrCyCtrl[arrCyNo.ElectValveName.AndeviationVacuum].Cmd.bOFF:=FALSE;	//正极纠偏台真空	
			DT_SingeMode();//单步选择	
			iEmptyFoldStep[1]:=1250;
		ELSE
			arrAxisCtrl[AxiseNo.AxisName.AnDTCarryingUpDown].Cmd.iGoSetPos:=2;//负极搬运升降2上升至凸轮耦合初始高度
		END_IF	
	END_IF	
1250://叠台搬运极片放回纠偏台
	IF NOT DP_SinStepe THEN
		IF arrAxisCtrl[AxiseNo.AxisName.AnDTCarryingUpDown].Cmd.arrbRealPoint[4] THEN
			arrAxisCtrl[AxiseNo.AxisName.AnDTCarryingUpDown].Cmd.iGoSetPos:=0;
			/// 吸盘破真空    纠偏台开真空
			Mach_Control.An_b.An_deviationFalg:=TRUE;//复位纠偏平台有料标记
			Mach_Control.An_b.An_DPCarryingFalg:=FALSE;//负极搬运真空吸盘有料标记复位
			Par.stDT_date.An_MQ_Slice[1]:=Par.stDT_date.An_MQ_Slice[2];
			DT_SingeMode();//单步选择	
			iEmptyFoldStep[1]:=1300;
		ELSE
			arrAxisCtrl[AxiseNo.AxisName.AnDTCarryingUpDown].Cmd.iGoSetPos:=4;//负极搬运升降2上升至凸轮耦合初始高度
		END_IF	
	END_IF			
1300:
	IF arrCyCtrl[arrCyNo.CylinderName.AnScrapbinCy].Status.ONState AND arrCyCtrl[arrCyNo.CylinderName.CaScrapbinUDCy].Status.OFFState AND
		arrCyCtrl[arrCyNo.CylinderName.CaScrapbinCy].Status.ONState AND arrCyCtrl[arrCyNo.CylinderName.PreDiaph].Status.OFFState AND 
		arrCyCtrl[arrCyNo.CylinderName.PoleHotCutterCy].Status.OFFState AND arrCyCtrl[arrCyNo.CylinderName.PoleTapeCy].Status.OFFState AND
		arrCyCtrl[arrCyNo.CylinderName.PoleTapeSplicerRCy].Status.ONState AND arrCyCtrl[arrCyNo.CylinderName.PoleTapeSplicerLCy].Status.ONState AND
        arrAxisCtrl[AxiseNo.AxisName.LeftYDUpDown].Cmd.arrbRealPoint[1] AND arrAxisCtrl[AxiseNo.AxisName.RightYDUpDown].Cmd.arrbRealPoint[1]  THEN
	     iEmptyFoldStep[1]:=2000;	
	END_IF	

	
	
	
1500://判断负极叠台搬运是否有片，有片的话放到纠偏台
	IF NOT DP_SinStepe THEN
		IF CA_CarryingPos1  THEN//负极搬运、叠片各轴在初始位
			IF arrCyCtrl[arrCyNo.ElectValveName.CaDTCarryingVacuum].Io.DIOnSwitch AND  Mach_Control.Ca_b.Ca_DPCarryingFalg THEN//正极再取片位且叠台搬运有片,把当前片放到纠偏台
				iEmptyFoldStep[1]:=1550;
			ELSE
				iEmptyFoldStep[1]:=3000;	
			END_IF
		ELSE
			IF (Ca_Step0=0 OR Ca_Step0=6666) AND (Ca_Step3=0 OR Ca_Step3=6666) AND Scan_TON[2].Q THEN
				Scan_TON[2].IN:=FALSE;		
				//DP_Step0:=9994;
				DTPosError[2]:=TRUE;
			END_IF
		END_IF
	END_IF	
1550://纠偏台回初始位
	//纠偏平台X1移动至初始位
	IF NOT DP_SinStepe THEN
		IF arrAxisCtrl[AxiseNo.AxisName.CadeviationX1].Status.Homed  AND arrAxisCtrl[AxiseNo.AxisName.CadeviationX1].Status.NoMoving AND NOT  arrAxisCtrl[AxiseNo.AxisName.CadeviationX1].Status.Error THEN
			IF arrAxisCtrl[AxiseNo.AxisName.CadeviationX1].Cmd.arrbRealPoint[1] THEN
				arrAxisCtrl[AxiseNo.AxisName.CadeviationX1].Cmd.iGoSetPos:=0;
			ELSE
				arrAxisCtrl[AxiseNo.AxisName.CadeviationX1].Cmd.iGoSetPos:=1;
			END_IF					
		END_IF
		//纠偏平台X2移动至初始位
		IF arrAxisCtrl[AxiseNo.AxisName.CadeviationX2].Status.Homed  AND arrAxisCtrl[AxiseNo.AxisName.CadeviationX2].Status.NoMoving AND NOT  arrAxisCtrl[AxiseNo.AxisName.CadeviationX2].Status.Error THEN
			IF arrAxisCtrl[AxiseNo.AxisName.CadeviationX2].Cmd.arrbRealPoint[1] THEN
				arrAxisCtrl[AxiseNo.AxisName.CadeviationX2].Cmd.iGoSetPos:=0;
			ELSE
				arrAxisCtrl[AxiseNo.AxisName.CadeviationX2].Cmd.iGoSetPos:=1;
			END_IF					
		END_IF
		//纠偏平台X2移动至初始位
		IF arrAxisCtrl[AxiseNo.AxisName.CadeviationY].Status.Homed  AND arrAxisCtrl[AxiseNo.AxisName.CadeviationY].Status.NoMoving AND NOT  arrAxisCtrl[AxiseNo.AxisName.CadeviationY].Status.Error THEN
			IF arrAxisCtrl[AxiseNo.AxisName.CadeviationY].Cmd.arrbRealPoint[1] THEN
				arrAxisCtrl[AxiseNo.AxisName.CadeviationY].Cmd.iGoSetPos:=0;
			ELSE
				arrAxisCtrl[AxiseNo.AxisName.CadeviationY].Cmd.iGoSetPos:=1;
			END_IF					
		END_IF
		IF arrAxisCtrl[AxiseNo.AxisName.CadeviationX1].Cmd.arrbRealPoint[1] AND arrAxisCtrl[AxiseNo.AxisName.CadeviationX2].Cmd.arrbRealPoint[1] AND arrAxisCtrl[AxiseNo.AxisName.CadeviationY].Cmd.arrbRealPoint[1] THEN
			DT_SingeMode();//单步选择	
			iEmptyFoldStep[1]:=1600;	
		END_IF	
	END_IF
1600:
	IF NOT DP_SinStepe THEN
		IF arrAxisCtrl[AxiseNo.AxisName.CaDTCarryingUpDown].Cmd.arrbRealPoint[3] THEN
			arrAxisCtrl[AxiseNo.AxisName.CaDTCarryingUpDown].Cmd.iGoSetPos:=0;
			/// 吸盘破真空    纠偏台开真空
			arrCyCtrl[arrCyNo.ElectValveName.CaDTCarryingVacuum].Cmd.bON:=TRUE;	//负极叠台搬运升降真空	真空
			arrCyCtrl[arrCyNo.ElectValveName.CaDTCarryingVacuum].Cmd.bOFF:=FALSE;	//负极叠台搬运升降真空破真空								
			arrCyCtrl[arrCyNo.ElectValveName.CadeviationVacuum].Cmd.bON:=TRUE;	//负极纠偏台真空			
			arrCyCtrl[arrCyNo.ElectValveName.CadeviationVacuum].Cmd.bOFF:=FALSE;	//负极纠偏台真空	   
			DT_SingeMode();//单步选择	
			iEmptyFoldStep[1]:=1650;
		ELSE
			arrAxisCtrl[AxiseNo.AxisName.CaDTCarryingUpDown].Cmd.iGoSetPos:=3;//负极搬运升降2上升至凸轮耦合初始高度
		END_IF	
	END_IF
1650://叠台搬运极片放回纠偏台
	IF NOT DP_SinStepe THEN
		IF arrAxisCtrl[AxiseNo.AxisName.CaDTCarryingUpDown].Cmd.arrbRealPoint[4] THEN
			arrAxisCtrl[AxiseNo.AxisName.CaDTCarryingUpDown].Cmd.iGoSetPos:=0;
			/// 吸盘破真空    纠偏台开真空
			Mach_Control.Ca_b.Ca_deviationFalg:=TRUE;//复位纠偏平台有料标记
			Mach_Control.Ca_b.Ca_DPCarryingFalg:=FALSE;//负极搬运真空吸盘有料标记复位
			Par.stDT_date.Ca_MQ_Slice[8]:=Par.stDT_date.Ca_MQ_Slice[9];
			DT_SingeMode();//单步选择	
			iEmptyFoldStep[1]:=1700;
		ELSE
			arrAxisCtrl[AxiseNo.AxisName.CaDTCarryingUpDown].Cmd.iGoSetPos:=4;//负极搬运升降2上升至凸轮耦合初始高度
		END_IF			
	END_IF	
1700:
	IF arrCyCtrl[arrCyNo.CylinderName.AnScrapbinCy].Status.ONState AND arrCyCtrl[arrCyNo.CylinderName.CaScrapbinUDCy].Status.OFFState AND
		arrCyCtrl[arrCyNo.CylinderName.CaScrapbinCy].Status.ONState AND arrCyCtrl[arrCyNo.CylinderName.PreDiaph].Status.OFFState AND 
		arrCyCtrl[arrCyNo.CylinderName.PoleHotCutterCy].Status.OFFState AND arrCyCtrl[arrCyNo.CylinderName.PoleTapeCy].Status.OFFState AND
		arrCyCtrl[arrCyNo.CylinderName.PoleTapeSplicerRCy].Status.ONState AND arrCyCtrl[arrCyNo.CylinderName.PoleTapeSplicerLCy].Status.ONState AND
        arrAxisCtrl[AxiseNo.AxisName.LeftYDUpDown].Cmd.arrbRealPoint[1] AND arrAxisCtrl[AxiseNo.AxisName.RightYDUpDown].Cmd.arrbRealPoint[1]  THEN
	     iEmptyFoldStep[1]:=3000;	
	END_IF	
	
	
		
2000:		
	IF NOT DP_SinStepe THEN
		IF AN_CarryingPos1  THEN//正极搬运、叠片各轴在初始位										
			IF CA_CarryingPos2 THEN//负极在叠片位
				IF arrAxisCtrl[AxiseNo.AxisName.SEPTATLine].Cmd.arrbRealPoint[1]  THEN
					DT_SingeMode();//单步选择	
					iEmptyFoldStep[1]:=2010;//
				ELSE
					Mach_Control.DT_b.Error[6]:=TRUE;//叠正极片凸轮耦合时，隔膜平移轴即不在负极叠片位，也不在正极叠片位报警
					//DP_Step0:=9998;
				END_IF;
			ELSIF  CA_CarryingPos1  THEN //负极取片位
				IF arrAxisCtrl[AxiseNo.AxisName.SEPTATLine].Cmd.arrbRealPoint[1]  THEN
					DT_SingeMode();//单步选择	
					iEmptyFoldStep[1]:=2030;//
				ELSIF arrAxisCtrl[AxiseNo.AxisName.SEPTATLine].Cmd.arrbRealPoint[2]  THEN
					DT_SingeMode();//单步选择	
					iEmptyFoldStep[1]:=2050;//
				ELSE
					Mach_Control.DT_b.Error[6]:=TRUE;//叠正极片凸轮耦合时，隔膜平移轴即不在负极叠片位，也不在正极叠片位报警
					//DP_Step0:=9999;
				END_IF;							
			ELSE
				Mach_Control.DT_b.Error[7]:=TRUE;//叠正极片凸轮耦合时，负极取片即不在取片位，也不在叠片位
				//DP_Step0:=10000;
			END_IF
		ELSE
			Mach_Control.DT_b.Error[8]:=TRUE;//叠正极片凸轮耦合时，正极片不在取片位
			//DP_Step0:=10001;
		END_IF
	END_IF		


2010://负极搬运、叠片各轴在初始位，隔膜平移轴负极叠片位、正极叠片在放极片初始位
	IF NOT DP_SinStepe THEN
		An_CanIn5:=TRUE;
		DT_SingeMode();//单步选择	
		iEmptyFoldStep[1]:=2020;	
	END_IF	
	
2020:
	IF NOT DP_SinStepe THEN
		IF NOT An_CanIn5 THEN
			DT_SingeMode();//单步选择	
			iEmptyFoldStep[1]:=2070;
		ELSIF fbAnCamInCarryingLine.bError  OR fbAnCamInDTCarryingLine.bError OR fbAnCamInDTCarryingUpDown.bError OR 
			fbAnCamInCarryingWhirling.bError OR fbCaCamInCarryingLine2.bError OR 
			fbCaCamInDTCarryingUpDown.bError OR fbCamInGMBuffer.bError OR fbCamInGMDanserMove.bError OR fbCamInVirGMDriver.bError   OR
			fbCamInRightYDUpDown.bError OR fbCamInRightYDLine.bError THEN
			An_CanIn5:=FALSE;
			Mach_Control.DT_b.Error[19]:=TRUE;//凸轮耦合报警
			//DP_Step0:=10004;		
		END_IF
	END_IF		
2030://负极搬运、叠片各轴在初始位，隔膜平移轴负极叠片位、正极叠片在取极片位
	IF NOT DP_SinStepe THEN
		DT_SingeMode();//单步选择	
		An_CanIn6:=TRUE;
		iEmptyFoldStep[1]:=2040;
	END_IF
2040:
	IF NOT DP_SinStepe THEN
		IF NOT An_CanIn6 THEN
			DT_SingeMode();//单步选择	
			iEmptyFoldStep[1]:=2070;
		ELSIF fbAnCamInCarryingLine.bError OR fbAnCamInDTCarryingLine.bError OR
			fbAnCamInDTCarryingUpDown.bError OR fbAnCamInCarryingWhirling.bError OR fbCamInGMBuffer.bError OR
			fbCamInGMDanserMove.bError OR fbCamInVirGMDriver.bError  OR fbCamInRightYDUpDown.bError OR
			fbCamInRightYDLine.bError THEN
			An_CanIn6:=FALSE;
			Mach_Control.DT_b.Error[19]:=TRUE;//凸轮耦合报警
			//DP_Step0:=10002;									
		END_IF
	END_IF
2050://负极搬运、叠片各轴在初始位，隔膜平移轴正极叠片位、正极叠片在取极片位
	IF NOT DP_SinStepe THEN
		An_CanIn7:=TRUE;
		DT_SingeMode();//单步选择	
		iEmptyFoldStep[1]:=2060;
	END_IF
2060:
	IF NOT DP_SinStepe THEN
		arrAxisCtrl[AxiseNo.VirAxisName.VirMain].Cmd	.bMoveAbs:=FALSE;	
		IF NOT An_CanIn7 THEN
			DT_SingeMode();//单步选择	
			iEmptyFoldStep[1]:=2070;
		ELSIF fbAnCamInCarryingLine.bError OR fbAnCamInCarryingUpDown.bError OR fbAnCamInDTCarryingLine.bError OR fbAnCamInDTCarryingUpDown.bError OR 
			fbAnCamInCarryingWhirling.bError OR fbCamInRightYDUpDown.bError OR fbCamInRightYDLine.bError THEN
			An_CanIn7:=FALSE;
			Mach_Control.DT_b.Error[19]:=TRUE;//凸轮耦合报警
			//DP_Step0:=10003;												
		END_IF
	END_IF	
	
2070://判断正极叠片搬运机械手上是否有极片
	VirMain_TON.IN:=FALSE;
	IF AN_CarryingPos1 THEN
		IF CA_CarryingPos1 THEN
			IF arrAxisCtrl[AxiseNo.AxisName.SEPTATLine].Cmd.arrbRealPoint[1]  THEN
				IF fbAnCamInCarryingLine.bInSync AND  fbAnCamInDTCarryingLine.bInSync AND
					fbAnCamInDTCarryingUpDown.bInSync AND fbAnCamInCarryingWhirling.bInSync AND fbCamInGMBuffer.bInSync AND
					fbCamInGMDanserMove.bInSync AND fbCamInVirGMDriver.bInSync  AND fbCamInRightYDUpDown.bInSync AND 
					fbCamInRightYDLine.bInSync  THEN
					iEmptyFoldStep[1]:=2071;
				
				END_IF
			ELSIF arrAxisCtrl[AxiseNo.AxisName.SEPTATLine].Cmd.arrbRealPoint[2]  THEN
				IF fbAnCamInCarryingLine.bInSync AND  fbAnCamInDTCarryingLine.bInSync AND fbAnCamInDTCarryingUpDown.bInSync  AND 
					fbAnCamInCarryingWhirling.bInSync AND fbCamInRightYDUpDown.bInSync AND fbCamInRightYDLine.bInSync THEN
					iEmptyFoldStep[1]:=2071;
				
				END_IF
			ELSE	
				Mach_Control.DT_b.Error[6]:=TRUE;//叠正极片凸轮耦合时，隔膜平移轴即不在负极叠片位，也不在正极叠片位报警
				//DP_Step0:=9999;
			END_IF	
		ELSIF CA_CarryingPos2 THEN
			IF arrAxisCtrl[AxiseNo.AxisName.SEPTATLine].Cmd.arrbRealPoint[1]  THEN
				IF fbAnCamInCarryingLine.bInSync AND fbAnCamInDTCarryingLine.bInSync AND fbAnCamInDTCarryingUpDown.bInSync AND 
					fbAnCamInCarryingWhirling.bInSync AND fbCaCamInCarryingLine2.bInSync AND fbCaCamInDTCarryingLine.bInSync AND
					fbCamInGMBuffer.bInSync AND fbCamInGMDanserMove.bInSync AND fbCamInVirGMDriver.bInSync   AND
					fbCamInRightYDUpDown.bInSync AND fbCamInRightYDLine.bInSync  THEN
					iEmptyFoldStep[1]:=2071;
				END_IF
			ELSE
				Mach_Control.DT_b.Error[6]:=TRUE;//叠正极片凸轮耦合时，隔膜平移轴即不在负极叠片位，也不在正极叠片位报警
				//DP_Step0:=9998;
			END_IF
		END_IF
	ELSE
		Mach_Control.DT_b.Error[8]:=TRUE;//叠正极片凸轮耦合时，正极片不在取片位
		//DP_Step0:=10001;
	END_IF
(*
	IF NOT DP_SinStepe THEN
		IF (NOT arrCyCtrl[arrCyNo.ElectValveName.AnDTCarryingVacuum].Io.DIOnSwitch AND NOT Mach_Control.An_b.An_DPCarryingFalg) THEN	
			DT_SingeMode();//单步选择	
			iEmptyFoldStep[1]:=2071;
		ELSE	
		  	Mach_Control.An_b.Error[28]:=TRUE; //正极叠片完空叠隔膜时，正极叠片搬运机械手真空有信号、标记有极片报警,请拿掉极片
		END_IF  
	END_IF
*)



3000:
	IF NOT DP_SinStepe THEN		
		Scan_TON[2].IN:=TRUE;	
		IF CA_CarryingPos1  THEN//负极搬运、叠片各轴在初始位
			Scan_TON[1].IN:=TRUE;	
			IF AN_CarryingPos2  THEN//正极在叠片位	
				IF arrAxisCtrl[AxiseNo.AxisName.SEPTATLine].Cmd.arrbRealPoint[2]   THEN													
					DT_SingeMode();//单步选择											
					iEmptyFoldStep[1]:=3010;//													
				ELSE
					Mach_Control.DT_b.Error[5]:=TRUE;//叠负极片凸轮耦合时，隔膜平移轴即不在负极叠片位，也不在正极叠片位报警
					//DP_Step0:=9991;	
				END_IF;
			ELSIF AN_CarryingPos1  THEN//在取片位																		
				IF arrAxisCtrl[AxiseNo.AxisName.SEPTATLine].Cmd.arrbRealPoint[1]  THEN
					DT_SingeMode();//单步选择										
					iEmptyFoldStep[1]:=3030;//
				ELSIF arrAxisCtrl[AxiseNo.AxisName.SEPTATLine].Cmd.arrbRealPoint[2] THEN
					DT_SingeMode();//单步选择										
					iEmptyFoldStep[1]:=3050;//
				ELSE
					Mach_Control.DT_b.Error[5]:=TRUE;//叠负极片凸轮耦合时，隔膜平移轴即不在负极叠片位，也不在正极叠片位报警
					//DP_Step0:=9992;	
				END_IF;							
			ELSIF Scan_TON[1].Q THEN
				Scan_TON[1].IN:=FALSE;	
				//DP_Step0:=9993;
				DTPosError[4]:=TRUE;
			END_IF
		ELSE
			IF (Ca_Step0=0 OR Ca_Step0=6666) AND (Ca_Step3=0 OR Ca_Step3=6666) AND Scan_TON[2].Q THEN
				Scan_TON[2].IN:=FALSE;		
				//DP_Step0:=9994;
				DTPosError[2]:=TRUE;
			END_IF
		END_IF
END_IF		

3010://负极搬运、叠片各轴在初始位，隔膜平移轴正极叠片位、正极叠片在放极片初始位
	IF NOT DP_SinStepe THEN
		Ca_CanIn5:=TRUE;
		DT_SingeMode();//单步选择	
		iEmptyFoldStep[1]:=3020;	
	END_IF
3020:
	IF NOT DP_SinStepe THEN
		arrAxisCtrl[AxiseNo.VirAxisName.VirMain].Cmd	.bMoveAbs:=FALSE;	
		IF NOT Ca_CanIn5 THEN
			DT_SingeMode();//单步选择	
			iEmptyFoldStep[1]:=3070;	
		ELSIF fbCaCamInCarryingLine2.bError OR  fbCaCamInDTCarryingLine.bError OR fbCaCamInDTCarryingUpDown.bError OR 
			fbCamInGMBuffer.bError OR fbCamInGMDanserMove.bError OR fbCamInVirGMDriver.bError OR fbAnCamInCarryingLine.bError OR 
			fbAnCamInDTCarryingLine.bError OR fbAnCamInCarryingWhirling.bError OR fbCamInLeftYDUpDown.bError OR fbCamInLeftYDLine.bError THEN
			Ca_CanIn5:=FALSE;
			Mach_Control.DT_b.Error[19]:=TRUE;//凸轮耦合报警
			//DP_Step0:=9998;										
		END_IF
	END_IF
3030://负极搬运、叠片各轴在初始位，隔膜平移轴负极叠片位、正极叠片在取极片位
	IF NOT DP_SinStepe THEN
		Ca_CanIn6:=TRUE;
		DT_SingeMode();//单步选择	
		iEmptyFoldStep[1]:=3040;
	END_IF
3040://判断凸轮耦合是否完成
	IF NOT DP_SinStepe THEN
		IF NOT Ca_CanIn6 THEN
			DT_SingeMode();//单步选择	
			iEmptyFoldStep[1]:=3070;
		ELSIF  fbCaCamInCarryingLine2.bError OR fbCaCamInDTCarryingLine.bError OR 
			fbCaCamInDTCarryingUpDown.bError OR fbCamInLeftYDUpDown.bError OR 	fbCamInLeftYDLine.bError THEN										
			Ca_CanIn6:=FALSE;
			Mach_Control.DT_b.Error[19]:=TRUE;//凸轮耦合报警
			//DP_Step0:=9995;		
		END_IF
	END_IF
3050://负极搬运、叠片各轴在初始位，隔膜平移轴正极叠片位、正极叠片在取极片位
	IF NOT DP_SinStepe THEN
		Ca_CanIn7:=TRUE;
		DT_SingeMode();//单步选择	
		iEmptyFoldStep[1]:=3060;
	END_IF
3060:
	IF NOT DP_SinStepe THEN
		arrAxisCtrl[AxiseNo.VirAxisName.VirMain].Cmd	.bMoveAbs:=FALSE;	
		IF NOT Ca_CanIn7 THEN
			DT_SingeMode();//单步选择																			
			iEmptyFoldStep[1]:=3070;
		ELSIF fbCaCamInCarryingLine2.bError OR fbCaCamInDTCarryingLine.bError OR 
			fbCaCamInDTCarryingUpDown.bError OR fbCamInGMBuffer.bError OR fbCamInGMDanserMove.bError OR
			fbCamInVirGMDriver.bError OR fbCamInLeftYDUpDown.bError OR fbCamInLeftYDLine.bError  THEN
			Ca_CanIn7:=FALSE;
			Mach_Control.DT_b.Error[19]:=TRUE;//凸轮耦合报警
			//DP_Step0:=9996;	
		END_IF
	END_IF

3070://判断负极叠片搬运机械手上是否有极片
	IF NOT DP_SinStepe THEN
		IF NOT arrCyCtrl[arrCyNo.ElectValveName.CaDTCarryingVacuum].Io.DIOnSwitch AND NOT Mach_Control.Ca_b.Ca_DPCarryingFalg  THEN	
			DT_SingeMode();//单步选择	
			iEmptyFoldStep[1]:=3071;
		ELSE	
		  	Mach_Control.Ca_b.Error[28]:=TRUE; //负极叠片完空叠隔膜时，负极叠片搬运机械手真空检测有信号报警,请拿掉极片
		END_IF  
	END_IF	 
3071://主轴启动
		arrAxisCtrl[AxiseNo.VirAxisName.VirMain].Cmd	.bDynamitcsParSel:=2;
		arrAxisPar[AxiseNo.VirAxisName.VirMain].fTagatTime:=VirMain_TagatTime;
		arrAxisCtrl[AxiseNo.VirAxisName.VirMain].Cmd	.fPositon_of_Abs:=360;
		arrAxisCtrl[AxiseNo.VirAxisName.VirMain].Cmd	.bMoveAbs:=TRUE;									
		IF  arrAxis[AxiseNo.VirAxisName.VirMain].Status.Moving AND arrAxisCtrl[AxiseNo.VirAxisName.VirMain].Status.fActPos>=10  THEN
			VirMain_TON.IN:=FALSE;
			arrAxisCtrl[AxiseNo.VirAxisName.VirMain].Cmd	.bMoveAbs:=FALSE;	
			iEmptyFoldStep[1]:=3080;	
		ELSE
			IF NOT VirMain_TON.Q THEN
				VirMain_TON.IN:=TRUE;
			ELSE
				VirMain_TON.IN:=FALSE;
				Mach_Control.DT_b.Error[22]:=TRUE;//主轴启动超时报警
				DP_Step0:=11006;	
			END_IF	
		END_IF	

		

END_CASE
END_IF

CASE iEmptyFoldStep[1] OF
2071://主轴启动
	
		arrAxisCtrl[AxiseNo.VirAxisName.VirMain].Cmd	.bDynamitcsParSel:=2;	
		arrAxisPar[AxiseNo.VirAxisName.VirMain].fTagatTime:=VirMain_TagatTime;
		arrAxisCtrl[AxiseNo.VirAxisName.VirMain].Cmd	.fPositon_of_Abs:=360;
		arrAxisCtrl[AxiseNo.VirAxisName.VirMain].Cmd	.bMoveAbs:=TRUE;	
		//fbCaCamInCarryingUpDown2OutCamFlge:=FALSE;//负极升降2凸轮解耦标记										
		IF  arrAxis[AxiseNo.VirAxisName.VirMain].Status.Moving AND arrAxisCtrl[AxiseNo.VirAxisName.VirMain].Status.fActPos>=10  THEN
			VirMain_TON.IN:=FALSE;
			arrAxisCtrl[AxiseNo.VirAxisName.VirMain].Cmd	.bMoveAbs:=FALSE;	
			iEmptyFoldStep[1]:=2080;	
		ELSE
			IF NOT VirMain_TON.Q THEN
				VirMain_TON.IN:=TRUE;
			ELSE
				VirMain_TON.IN:=FALSE;
				Mach_Control.DT_b.Error[22]:=TRUE;//主轴启动超时报警
				DP_Step0:=11006;	
			END_IF	
		END_IF	
2080:
	IF arrAxis[AxiseNo.VirAxisName.VirMain].NcToPlc.SetPos=360 AND  arrAxis[AxiseNo.VirAxisName.VirMain].Status.NotMoving  THEN
		Mach_Control.An_b.An_FirstFoldCnt:=Mach_Control.An_b.An_FirstFoldCnt+1;
		DPcount:=DPcount+1;		
		DP_Step1:=100;//解除耦合，主轴回零子程序
		//arrAxisCtrl[AxiseNo.AxisName.DTUpDown].Cmd.fPosition_of_Rel:=-Par.stDT_date.SEPTA_Thickness;
		//arrAxisPar[AxiseNo.AxisName.DTUpDown].fVelocity_of_Rel:=100;
		//arrAxisCtrl[AxiseNo.AxisName.DTUpDown].Cmd.bMoveRel:=TRUE;
		iEmptyFoldStep[1]:=2100;
	END_IF
2100://判断首层隔膜是否完成
	IF  Mach_Control.An_b.An_FirstFoldCnt=Mach_Control.An_b.An_FirstFoldSet  AND Mach_Control.An_b.An_FirstFoldSet<>0
	(*AND Mach_Control.Ca_b.Ca_FirstFoldCnt=Mach_Control.Ca_b.Ca_FirstFoldSet AND Mach_Control.Ca_b.Ca_FirstFoldSet<>0 *)THEN 
		bFirstFoldFinish[1]:=TRUE;//首层隔膜空叠完成
		iEmptyFoldStep[1]:=0;
		DP_Step0:=0;
		 CCD.Over.Finish.OverhandResult:=0;	
	ELSE
		bFirstFoldFinish[1]:=FALSE;//首层隔膜空叠完成
		iEmptyFoldStep[1]:=100;
	END_IF
	
	
	
	
	
3080:
	IF arrAxis[AxiseNo.VirAxisName.VirMain].NcToPlc.SetPos=360 AND  arrAxis[AxiseNo.VirAxisName.VirMain].Status.NotMoving  THEN
		Mach_Control.Ca_b.Ca_FirstFoldCnt:=Mach_Control.Ca_b.Ca_FirstFoldCnt+1;
		DPcount:=DPcount+1;		
		DP_Step1:=100;//解除耦合，主轴回零子程序
		//arrAxisCtrl[AxiseNo.AxisName.DTUpDown].Cmd.fPosition_of_Rel:=-Par.stDT_date.SEPTA_Thickness;
		//arrAxisPar[AxiseNo.AxisName.DTUpDown].fVelocity_of_Rel:=100;
		//arrAxisCtrl[AxiseNo.AxisName.DTUpDown].Cmd.bMoveRel:=TRUE;							
		iEmptyFoldStep[1]:=3100;
	END_IF	
3100:
	IF  Mach_Control.An_b.An_FirstFoldCnt=Mach_Control.An_b.An_FirstFoldSet  AND Mach_Control.An_b.An_FirstFoldSet<>0
	AND Mach_Control.Ca_b.Ca_FirstFoldCnt=Mach_Control.Ca_b.Ca_FirstFoldSet AND Mach_Control.Ca_b.Ca_FirstFoldSet<>0 THEN 
		bFirstFoldFinish[1]:=TRUE;//首层隔膜空叠完成
		iEmptyFoldStep[1]:=0;
		DP_Step0:=0;
		 CCD.Over.Finish.OverhandResult:=0;	
	ELSE
		bFirstFoldFinish[1]:=FALSE;//首层隔膜空叠完成
		iEmptyFoldStep[1]:=100;
	END_IF		
END_CASE	


//判断运动过程中的耦合状态,若核膜平移轴未动作则停止主轴
IF iEmptyFoldStep[1]=2080 THEN
	IF arrAxis[AxiseNo.VirAxisName.VirMain].Status.Moving AND arrAxisCtrl[AxiseNo.VirAxisName.VirMain].Status.fActPos>=20 AND arrAxisCtrl[AxiseNo.VirAxisName.VirMain].Status.fActPos<=245  THEN
		IF (NOT fbCamInGMDanserMove.bInSync OR NOT arrAxis[AxiseNo.AxisName.SEPTATLine].Status.Moving ) AND NOT  arrAxisCtrl[AxiseNo.AxisName.SEPTATLine].Cmd.arrbRealPoint[2] THEN  
			arrAxisCtrl[AxiseNo.VirAxisName.VirMain].Cmd. bStop:=TRUE;	
			Mach_Control.DT_b.Error[55]:=TRUE;//叠首层隔膜过程中，隔膜平移轴未动作
		ELSE
			arrAxisCtrl[AxiseNo.VirAxisName.VirMain].Cmd. bStop:=FALSE;	
		END_IF
	END_IF
END_IF
END_ACTION

ACTION GMEmptyFold2:
;//叠完电芯的空叠自动步	iEmptyFoldStep[2]
END_ACTION

ACTION GMEmptyFold3:
;//蓝胶、黄标空叠自动步		iEmptyFoldStep[3]
END_ACTION

ACTION Manual:
pt_Time:=T#0.5S;
//负极缓存皮带末端破真空打开后延时0.5S复位
(*
arTON[0](IN:=arrCyCtrl[arrCyNo.ElectValveName.CaLoadUpBeltVacuumBark].Status.ONState , PT:=pt_Time , Q=> , ET=> );
IF arTON[0].Q THEN
	arrCyCtrl[arrCyNo.ElectValveName.CaLoadUpBeltVacuumBark].Cmd.bOFF:=TRUE;
END_IF
*)
//负极搬运2破真空真打开后，延时0.5S关闭
arTON[1](IN:=arrCyCtrl[arrCyNo.ElectValveName.CaCarryingVacuumBark2].Status.ONState , PT:=pt_Time , Q=> , ET=> );
IF arTON[1].Q THEN
	arrCyCtrl[arrCyNo.ElectValveName.CaCarryingVacuumBark2].Cmd.bOFF:=TRUE;
	arrCyCtrl[arrCyNo.ElectValveName.CaCarryingVacuumBark2].Cmd.bON:=FALSE;
END_IF
//负极叠片搬运升降破真空打开后延时0.5S关闭
arTON[2](IN:=arrCyCtrl[arrCyNo.ElectValveName.CaDTCarryingVacuumBark].Status.ONState , PT:=pt_Time , Q=> , ET=> );
IF arTON[2].Q THEN
	arrCyCtrl[arrCyNo.ElectValveName.CaDTCarryingVacuumBark].Cmd.bOFF:=TRUE;
	arrCyCtrl[arrCyNo.ElectValveName.CaDTCarryingVacuumBark].Cmd.bOn:=FALSE;
END_IF



//负极纠偏平台破真空打开后延时0.5S复位
arTON[3](IN:=arrCyCtrl[arrCyNo.ElectValveName.CadeviationVacuumBark].Status.ONState , PT:=pt_Time , Q=> , ET=> );
IF arTON[3].Q THEN
	arrCyCtrl[arrCyNo.ElectValveName.CadeviationVacuumBark].Cmd.bOFF:=TRUE;
	arrCyCtrl[arrCyNo.ElectValveName.CadeviationVacuumBark].Cmd.bON:=FALSE;
END_IF




(*
//正极模切送料分段皮带破真空打开后延时0.5S关闭
arTON[4](IN:=arrCyCtrl[arrCyNo.ElectValveName.AnBeltVacuumBark].Status.ONState , PT:=pt_Time , Q=> , ET=> );
IF arTON[4].Q THEN
	arrCyCtrl[arrCyNo.ElectValveName.AnBeltVacuumBark].Cmd.bOFF:=TRUE;
END_IF
*)
//正极叠片搬运升降破真空打开后延时0.5S关闭
arTON[5](IN:=arrCyCtrl[arrCyNo.ElectValveName.AnDTCarryingVacuumBark].Status.ONState , PT:=pt_Time , Q=> , ET=> );
IF arTON[5].Q THEN
	arrCyCtrl[arrCyNo.ElectValveName.AnDTCarryingVacuumBark].Cmd.bOFF:=TRUE;
	arrCyCtrl[arrCyNo.ElectValveName.AnDTCarryingVacuumBark].Cmd.bON:=FALSE;
END_IF
//正极纠偏平台破真空打开后延时0.5S关闭
arTON[6](IN:=arrCyCtrl[arrCyNo.ElectValveName.AndeviationVacuumBark].Status.ONState , PT:=pt_Time , Q=> , ET=> );
IF arTON[6].Q THEN
	arrCyCtrl[arrCyNo.ElectValveName.AndeviationVacuumBark].Cmd.bOFF:=TRUE;
	arrCyCtrl[arrCyNo.ElectValveName.AndeviationVacuumBark].Cmd.bON:=FALSE;
END_IF
//正极送片搬运破真空打开后延时关闭
arTON[7](IN:=arrCyCtrl[arrCyNo.ElectValveName.AnCarryingVacuumBark].Status.ONState , PT:=pt_time , Q=> , ET=> );
IF arTON[7].Q THEN
	arrCyCtrl[arrCyNo.ElectValveName.AnCarryingVacuumBark].Cmd.bOFF:=TRUE;
	arrCyCtrl[arrCyNo.ElectValveName.AnCarryingVacuumBark].Cmd.bON:=FALSE;
END_IF
(*
//负极送片皮带破真空打开后延时关闭
arTON[8](IN:=arrCyCtrl[arrCyNo.ElectValveName.CaLoadUpBeltVacuumBark].Status.ONState , PT:=pt_time , Q=> , ET=> );
IF arTON[8].Q THEN
	arrCyCtrl[arrCyNo.ElectValveName.CaLoadUpBeltVacuumBark].Cmd.bOFF:=TRUE;
END_IF
*)
(*
//负极模切皮带破真空打开后延时关闭
arTON[9](IN:=arrCyCtrl[arrCyNo.ElectValveName.CaMQBeltVacuumBark].Status.ONState , PT:=pt_time , Q=> , ET=> );
IF arTON[9].Q THEN
	arrCyCtrl[arrCyNo.ElectValveName.CaMQBeltVacuumBark].Cmd.bOFF:=TRUE;
END_IF
*)

//负极送片皮带破真空打开后延时关闭
arTON[10](IN:=arrCyCtrl[arrCyNo.ElectValveName.CaCarryingVacuumBark1].Status.ONState , PT:=pt_time , Q=> , ET=> );
IF arTON[10].Q THEN
	arrCyCtrl[arrCyNo.ElectValveName.CaCarryingVacuumBark1].Cmd.bOFF:=TRUE;
END_IF

//气胀轴手动
rPoleIn_btn(CLK:=Mach_Control.btn.PoleInflationbtn , Q=> );
IF NOT arrCyCtrl[arrCyNo.CylinderName.PoleInflationCy].Status.OFFState AND rPoleIn_btn.Q  THEN
	arrCyCtrl[arrCyNo.CylinderName.PoleInflationCy].Cmd.bOFF:=TRUE;
ELSIF NOT arrCyCtrl[arrCyNo.CylinderName.PoleInflationCy].Status.ONState AND rPoleIn_btn.Q  THEN 
	arrCyCtrl[arrCyNo.CylinderName.PoleInflationCy].Cmd.bON:=TRUE;
END_IF
//气胀轴按钮灯
Mach_Control.btn.PoleInflationLights:=arrCyCtrl[arrCyNo.CylinderName.PoleInflationCy].Status.ONState;
//左压隔膜手动
rPoleTapeL_btn(CLK:=Mach_Control.btn.PoleTapeSplicerLbtn , Q=> );
IF NOT arrCyCtrl[arrCyNo.CylinderName.PoleTapeSplicerLCy].Status.OFFState AND rPoleTapeL_btn.Q  THEN
	arrCyCtrl[arrCyNo.CylinderName.PoleTapeSplicerLCy].Cmd.bOFF:=TRUE;
ELSIF NOT arrCyCtrl[arrCyNo.CylinderName.PoleTapeSplicerLCy].Status.ONState AND rPoleTapeL_btn.Q  THEN 
	arrCyCtrl[arrCyNo.CylinderName.PoleTapeSplicerLCy].Cmd.bON:=TRUE;
END_IF
//左压隔膜按钮灯
Mach_Control.btn.PoleInflationLights:=arrCyCtrl[arrCyNo.CylinderName.PoleTapeSplicerLCy].Status.ONState;
//右压隔膜手动
rPoleTapeR_btn(CLK:=Mach_Control.btn.PoleTapeSplicerRbtn , Q=> );
IF NOT arrCyCtrl[arrCyNo.CylinderName.PoleTapeSplicerRCy].Status.OFFState AND rPoleTapeR_btn.Q  THEN
	arrCyCtrl[arrCyNo.CylinderName.PoleTapeSplicerRCy].Cmd.bOFF:=TRUE;
ELSIF NOT arrCyCtrl[arrCyNo.CylinderName.PoleTapeSplicerRCy].Status.ONState AND rPoleTapeR_btn.Q  THEN 
	arrCyCtrl[arrCyNo.CylinderName.PoleTapeSplicerRCy].Cmd.bON:=TRUE;
END_IF
//右压隔膜灯
Mach_Control.btn.PoleTapeSplicerLLights:=arrCyCtrl[arrCyNo.CylinderName.PoleTapeSplicerRCy].Status.ONState;
//压二维码胶气缸手动
rCodeGluePressCy_btn(CLK:=Mach_Control.btn.codeGluePressbtn , Q=> );
IF NOT arrCyCtrl[arrCyNo.CylinderName.CodeGluePressCy].Status.OFFState AND rCodeGluePressCy_btn.Q THEN
	arrCyCtrl[arrCyNo.CylinderName.CodeGluePressCy].Cmd.bOFF:=TRUE;
ELSIF NOT arrCyCtrl[arrCyNo.CylinderName.CodeGluePressCy].Status.ONState AND rCodeGluePressCy_btn.Q THEN 
	arrCyCtrl[arrCyNo.CylinderName.CodeGluePressCy].Cmd.bON:=TRUE;
END_IF
//压二维码胶灯
Mach_Control.btn.codeGlueLights:=arrCyCtrl[arrCyNo.CylinderName.CodeGluePressCy].Cmd.bON;
//压蓝胶气缸手动
rGluePressCy_btn(CLK:=Mach_Control.btn.BlueGluePressbtn , Q=> );
IF NOT arrCyCtrl[arrCyNo.CylinderName.GluePressCy].Status.OFFState AND rGluePressCy_btn.Q THEN
	arrCyCtrl[arrCyNo.CylinderName.GluePressCy].Cmd.bOFF:=TRUE;
ELSIF NOT arrCyCtrl[arrCyNo.CylinderName.GluePressCy].Status.ONState AND rGluePressCy_btn.Q THEN
	arrCyCtrl[arrCyNo.CylinderName.GluePressCy].Cmd.bON:=TRUE;
END_IF
//压蓝胶灯
Mach_Control.btn.BlueGlueLights:=arrCyCtrl[arrCyNo.CylinderName.GluePressCy].Status.ONState;


//正极防撞感应信号，停止叠片搬运平移
AnAxisbstop_R(CLK:= arrAxisbstop[AxiseNo.AxisName.AnDTCarryingLine] , Q=> );//HMI轴停止上升沿
AnAxisbstop_F(CLK:= arrAxisbstop[AxiseNo.AxisName.AnDTCarryingLine] , Q=> );//HMI轴停止下降沿

IF AnAxisbstop_R.Q AND Mach_Control.U.DT_iMode=3 THEN 
   arrAxisCtrl[AxiseNo.AxisName.AnDTCarryingLine].Cmd.bStop:=TRUE;
END_IF
 
IF AnAxisbstop_F.Q AND Mach_Control.U.DT_iMode=3 THEN 
   arrAxisCtrl[AxiseNo.AxisName.AnDTCarryingLine].Cmd.bStop:=FALSE;
END_IF

AnAxisbstop1_R(CLK:= arrAxisbstop[AxiseNo.AxisName.AnCarryingLine] , Q=> );//HMI轴停止上升沿
AnAxisbstop1_F(CLK:= arrAxisbstop[AxiseNo.AxisName.AnCarryingLine] , Q=> );//HMI轴停止下降沿

IF AnAxisbstop1_R.Q AND Mach_Control.U.DT_iMode=3 THEN 
   arrAxisCtrl[AxiseNo.AxisName.AnCarryingLine].Cmd.bStop:=TRUE;
END_IF
 
IF AnAxisbstop1_F.Q AND Mach_Control.U.DT_iMode=3 THEN 
   arrAxisCtrl[AxiseNo.AxisName.AnCarryingLine].Cmd.bStop:=FALSE;
END_IF

IF NOT Mach_Control.se.AnLimitSwitch AND arrAxisCtrl[AxiseNo.AxisName.AnCarryingLine].Status.Homed AND arrAxisCtrl[AxiseNo.AxisName.AnDTCarryingLine].Status.Homed AND 
NOT arrAxis[AxiseNo.AxisName.AnDTCarryingLine].Status.Coupled AND arrAxis[AxiseNo.VirAxisName.VirMain].Status.NotMoving THEN
	arrAxisCtrl[AxiseNo.AxisName.AnDTCarryingLine].Cmd.bStop:=TRUE;
	Mach_Control.An_b.Error[14]:=TRUE;//正极防撞感应信号报警
END_IF
//负极防撞感应信号，停止负极搬运平移
CaAxisbstop_R(CLK:= arrAxisbstop[AxiseNo.AxisName.CaDTCarryingLine] , Q=> );//HMI轴停止上升沿
CaAxisbstop_F(CLK:= arrAxisbstop[AxiseNo.AxisName.CaDTCarryingLine] , Q=> );//HMI轴停止下降沿

IF CaAxisbstop_R.Q AND Mach_Control.U.DT_iMode=3 THEN 
   arrAxisCtrl[AxiseNo.AxisName.CaDTCarryingLine].Cmd.bStop:=TRUE;
END_IF
 
IF CaAxisbstop_F.Q AND Mach_Control.U.DT_iMode=3 THEN 
   arrAxisCtrl[AxiseNo.AxisName.CaDTCarryingLine].Cmd.bStop:=FALSE;
END_IF

CaAxisbstop1_R(CLK:= arrAxisbstop[AxiseNo.AxisName.CaCarryingLine2] , Q=> );//HMI轴停止上升沿
CaAxisbstop1_F(CLK:= arrAxisbstop[AxiseNo.AxisName.CaCarryingLine2] , Q=> );//HMI轴停止下降沿

IF CaAxisbstop1_R.Q AND Mach_Control.U.DT_iMode=3 THEN 
   arrAxisCtrl[AxiseNo.AxisName.CaCarryingLine2].Cmd.bStop:=TRUE;
END_IF
 
IF CaAxisbstop1_F.Q AND Mach_Control.U.DT_iMode=3 THEN 
   arrAxisCtrl[AxiseNo.AxisName.CaCarryingLine2].Cmd.bStop:=FALSE;
END_IF

IF NOT Mach_Control.se.CaLimitSwitch AND arrAxisCtrl[AxiseNo.AxisName.CaCarryingLine2].Status.Homed AND arrAxisCtrl[AxiseNo.AxisName.CaDTCarryingLine].Status.Homed AND
   NOT arrAxis[AxiseNo.AxisName.CaDTCarryingLine].Status.Coupled AND arrAxis[AxiseNo.VirAxisName.VirMain].Status.NotMoving THEN
	arrAxisCtrl[AxiseNo.AxisName.CaDTCarryingLine].Cmd.bStop:=TRUE;
	Mach_Control.Ca_b.Error[17]:=TRUE;//负极防撞感应信报警
END_IF
//急停
IF NOT Mach_Control.btn.EmStopbtn1 THEN
								
								Ca_Step0:=0;//负极搬运子程序1
								Ca_Step1:=0;//负极搬运子程序2
								Ca_Step2:=0;//负极搬运子程序3
								Ca_Step3:=0;//负极搬运子程序4
								Ca_RectifydevStep :=0;//纠偏自动程序
								Ca_Demarcate_Step0:=0;//纠偏标定程序步
								Ca_RecdevPla_Step0:=0;//纠偏自动程序步
								Ca_StandbyStep0:=0;//负极自动备料自动步清零
								Ca_StandbyStep1:=0;//叠负极片，判断真空阀的开关
								Ca_StandbyStep2:=0;
								Ca_StandbyStep4:=0;
								Ca_StandbyStep5:=0;//叠负极片，判断主轴是否完成
								Step_InitCaDT:=0;//取负极片回原点
								Step_InitCaDT0:=0;//负极皮带流水线
								Ca_GohomeDone:=FALSE;
								Ca_BeltGohomeDone:=FALSE;
								
								An_StandbyStep0:=0;//正极纠偏平台自动步
								An_StandbyStep1:=0;//正极取片备料步清零
								An_StandbyStep2:=0;//叠正极片，判断真空、破真空
								An_StandbyStep3:=0;//叠正极片，判断主轴是否完成
								An_Step0:=0;//正极取片子程序1
								An_Step1:=0;//正极取片子程序2
								An_Step2:=0;//正极取片子程序3
								An_Step3:=0;//正极取片子程序4
								An_Demarcate_Step0:=0;//正极标定自动程序
								An_RecdevPla_Step0:=0;	
								An_GohomeDone:=FALSE;

								
		                     	Ca_OverNGStep:=0;	
	                			An_OverNGStep:=0;									
								DP_Step0:=0;
								DP_Step1:=0;	
								DP_Step3:=0;
								DP_Step4:=0;
								Mach_Control.DT_b.OffloadRequest:=FALSE;//叠电芯完成，请求下电芯
								Step_InitDT:=0;
								DTIniti_Done:=FALSE;
								Dietai_GohomeDone:=FALSE;
								arrAxisCtrl[AxiseNo.VirAxisName.VirMain].Cmd	.bStop:=TRUE;//主轴停止
								
								
								WZIniti_Done:=FALSE;//初始化完成	
								TailCurlStep3 :=0;
								TailCurlStep4:=0;
								TailCurlStep5:=0;
								TailCurlStart:=FALSE;//复位尾卷启动
								Mach_Control.WJ_b.TailCurlDone	:=FALSE;	//尾卷完成
								arrAxisCtrl[AxiseNo.VirAxisName.VirTailCurl].Cmd.bStop:=TRUE;//主轴停止
								tTailCurlTON.IN:=FALSE;
								TailCurlStep1:=0;		
								WZIniti_Done:=FALSE;
								Tailcurl_GohomeDone:=FALSE;
								
								StickerStep0:=0;
								Sticker_Step0:=0;
								Sticker_Step1:=0;
								TJIniti_Done:=FALSE;
								Sticker_GohomeDone:=FALSE;
END_IF


IF Mach_Control.U.DT_iMode=3 AND arrCyCtrl[arrCyNo.CylinderName.PoleInflationCy].Status.OFFState AND arrAxisCtrl[AxiseNo.AxisName.SEPTAdeviation1].Status.Homed 
	AND arrAxisCtrl[AxiseNo.AxisName.SEPTAdeviation2].Status.Homed AND NOT Pole_BJ THEN
	IF 	arrAxisCtrl[AxiseNo.AxisName.SEPTAdeviation1].Status.Homed AND arrAxisCtrl[AxiseNo.AxisName.SEPTAdeviation1].Status.NoMoving THEN
		IF arrAxisCtrl[AxiseNo.AxisName.SEPTAdeviation1].Cmd.arrbRealPoint[1] THEN
			arrAxisCtrl[AxiseNo.AxisName.SEPTAdeviation1].Cmd.iGoSetPos:=0;
		ELSE
			arrAxisCtrl[AxiseNo.AxisName.SEPTAdeviation1].Cmd.iGoSetPos:=1;
		END_IF
	END_IF	
	IF 	arrAxisCtrl[AxiseNo.AxisName.SEPTAdeviation2].Status.Homed AND arrAxisCtrl[AxiseNo.AxisName.SEPTAdeviation2].Status.NoMoving THEN
		IF arrAxisCtrl[AxiseNo.AxisName.SEPTAdeviation2].Cmd.arrbRealPoint[1] THEN
			arrAxisCtrl[AxiseNo.AxisName.SEPTAdeviation2].Cmd.iGoSetPos:=0;
		ELSE
			arrAxisCtrl[AxiseNo.AxisName.SEPTAdeviation2].Cmd.iGoSetPos:=1;
		END_IF
	END_IF
	IF arrAxisCtrl[AxiseNo.AxisName.SEPTAdeviation1].Status.Homed AND arrAxisCtrl[AxiseNo.AxisName.SEPTAdeviation2].Status.Homed 
	AND arrAxisCtrl[AxiseNo.AxisName.SEPTAdeviation1].Cmd.arrbRealPoint[1] AND arrAxisCtrl[AxiseNo.AxisName.SEPTAdeviation2].Cmd.arrbRealPoint[1] THEN
		Pole_BJ:=TRUE;
	END_IF
END_IF

IF arrCyCtrl[arrCyNo.CylinderName.PoleInflationCy].Status.ONState OR NOT arrCyCtrl[arrCyNo.CylinderName.PoleInflationCy].Status.OFFState THEN
	Pole_BJ:=FALSE;
END_IF


//压刀高度计算
arrAxisPar[AxiseNo.AxisName.LeftYDUpDown].arrTargetPoint[14]:=arrAxisPar[AxiseNo.AxisName.LeftYDUpDown].arrTargetPoint[1]-arrAxisPar[AxiseNo.AxisName.LeftYDUpDown].arrTargetPoint[11]-arrAxisPar[AxiseNo.AxisName.LeftYDUpDown].arrTargetPoint[13];
arrAxisPar[AxiseNo.AxisName.LeftYDUpDown].arrTargetPoint[15]:=arrAxisPar[AxiseNo.AxisName.LeftYDUpDown].arrTargetPoint[1]-arrAxisPar[AxiseNo.AxisName.LeftYDUpDown].arrTargetPoint[12]-arrAxisPar[AxiseNo.AxisName.LeftYDUpDown].arrTargetPoint[13];
arrAxisPar[AxiseNo.AxisName.RightYDUpDown].arrTargetPoint[14]:=arrAxisPar[AxiseNo.AxisName.RightYDUpDown].arrTargetPoint[1]-arrAxisPar[AxiseNo.AxisName.RightYDUpDown].arrTargetPoint[11]-arrAxisPar[AxiseNo.AxisName.RightYDUpDown].arrTargetPoint[13];
arrAxisPar[AxiseNo.AxisName.RightYDUpDown].arrTargetPoint[15]:=arrAxisPar[AxiseNo.AxisName.RightYDUpDown].arrTargetPoint[1]-arrAxisPar[AxiseNo.AxisName.RightYDUpDown].arrTargetPoint[12]-arrAxisPar[AxiseNo.AxisName.RightYDUpDown].arrTargetPoint[13];

//夹膜夹板气缸条件
IF  arrAxisCtrl[AxiseNo.AxisName.TailCurlLine].Cmd.arrbRealPoint[1] 
OR  arrAxisCtrl[AxiseNo.AxisName.TailCurlLine].Cmd.arrbRealPoint[5]
OR Mach_Control.U.WJ_iMode=1 THEN
	arrCyCtrl[arrCyNo.CylinderName.	PoleSplintCy_U].Cmd.OnCondition:=TRUE;
	arrCyCtrl[arrCyNo.CylinderName.	PoleSplintCy_D].Cmd.OnCondition:=TRUE;
ELSE
	arrCyCtrl[arrCyNo.CylinderName.	PoleSplintCy_U].Cmd.OnCondition:=FALSE;
	arrCyCtrl[arrCyNo.CylinderName.	PoleSplintCy_D].Cmd.OnCondition:=FALSE;
END_IF
END_ACTION

ACTION ModeENLimk:
//屏蔽链接
Mach_Control.DT_b.FirstEmpFold:=par.iModeEN.FirstEmpFoldEN;				//首层空叠隔膜屏蔽
Mach_Control.DT_b.DP_Mode:=NOT par.iModeEN.DP_ModeEN;				//尾层空叠隔膜屏蔽
Mach_Control.DT_b.RectifydevModel:=par.iModeEN.RectifydevModelEN;			//隔膜纠偏屏蔽
Mach_Control.U.EmptyRunMode:=par.iModeEN.EmptyRunModeEN;				//空叠隔膜屏蔽
Mach_Control.U.CCD_ChosesHMI:=par.iModeEN.CCD_ChosesHMIEN;			//CCD屏蔽
Mach_Control.DT_b.DT_CCD_TwoModel:=NOT par.iModeEN.DT_CCD_TwoModelEN;		//CCD复检屏蔽
Mach_Control.DT_b.DT_Overhang:=par.iModeEN.DT_OverhangEN;				//对齐度屏蔽
Mach_Control.DT_b.DT_CellNG_TF:=NOT par.iModeEN.DT_CellNG_TFEN;				//对齐度踢废屏蔽 
Mach_Control.DT_b.DT_OHclosure:= par.iModeEN.DT_OHclosureEN;				//对齐度闭环屏蔽		ON是屏蔽
Mach_Control.DT_b.GMAngleALMsel:= par.iModeEN.GMAngleALMsel; //隔膜卷径报警屏蔽		ON是屏蔽
END_ACTION

ACTION MotionCoe_Write:

//nSlaveAddr :ARRAY[1..6] OF INT :=[1003,1008,1018,1019,1020,1021] ;     //EtherCAT支路驱动器ID

//'192.168.10.10.4.1'	EtherCat支路ID
(*
//隔膜平移地址
P2M1_Par.stDT_date.EtherCatAddr[1]:=1172;
P2M2_Par.stDT_date.EtherCatAddr[1]:=1123;
P2M3_Par.stDT_date.EtherCatAddr[1]:=1077;

//隔膜缓存地址
P2M1_Par.stDT_date.EtherCatAddr[2]:=1173;
P2M2_Par.stDT_date.EtherCatAddr[2]:=1124;
P2M3_Par.stDT_date.EtherCatAddr[2]:=1078;

//正极送片搬运平移地址
P2M1_Par.stDT_date.EtherCatAddr[3]:=1170;
P2M2_Par.stDT_date.EtherCatAddr[3]:=1121;
P2M3_Par.stDT_date.EtherCatAddr[3]:=1075;

//正极叠片搬运平移地址
P2M1_Par.stDT_date.EtherCatAddr[4]:=1171;
P2M2_Par.stDT_date.EtherCatAddr[4]:=1122;
P2M3_Par.stDT_date.EtherCatAddr[4]:=1076;

//负极送片搬运平移地址
P2M1_Par.stDT_date.EtherCatAddr[5]:=1188;
P2M2_Par.stDT_date.EtherCatAddr[5]:=1139;
P2M3_Par.stDT_date.EtherCatAddr[5]:=1093;

//负极叠片搬运平移地址
P2M1_Par.stDT_date.EtherCatAddr[6]:=1172;
P2M2_Par.stDT_date.EtherCatAddr[6]:=1140;
P2M3_Par.stDT_date.EtherCatAddr[6]:=1094;

//////////////////////////////////////////////////////////////////////一号叠台隔膜平移
FB_EcCoESdoWrite_SEPTATLine[1](
	sNetId:= '192.168.10.10.4.1', 
	nSlaveAddr:=Par.stDT_date.EtherCatAddr[1] ,   //隔膜平移
	nSubIndex:=0 , 
	nIndex:=16#2108 ,   //  平滑时间
	pSrcBuf:=ADR(Par.stDT_date.SEPTATLine_fSmoothValue[1]),       //写入参数值 
	cbBufLen:=SIZEOF(Par.stDT_date.SEPTATLine_fSmoothValue[1]),    
	bExecute:= Par.stDT_date.SEPTATLine_bWriteCoeValue[1],    
	tTimeout:= T#3S, 
	bBusy=> , 
	bError=> , 
	nErrId=> );
	
FB_EcCoESdoWrite_SEPTATLine[2](
	sNetId:='192.168.10.10.4.1', 
	nSlaveAddr:=Par.stDT_date.EtherCatAddr[1] ,   //隔膜平移
	nSubIndex:=0 , 
	nIndex:=16#2109 ,   // 平滑方式
	pSrcBuf:=ADR(Par.stDT_date.SEPTATLine_fSmoothValue[2]),       //写入参数值 
	cbBufLen:=SIZEOF(Par.stDT_date.SEPTATLine_fSmoothValue[2]),    
	bExecute:= Par.stDT_date.SEPTATLine_bWriteCoeValue[2],    
	tTimeout:= T#3S, 
	bBusy=> , 
	bError=> , 
	nErrId=> );

//平滑时间参数保存	
FB_EcCoESdoWrite_SEPTATLine[3](
	sNetId:= '192.168.10.10.4.1', 
	nSlaveAddr:=Par.stDT_date.EtherCatAddr[1] ,   //隔膜平移
	nSubIndex:=0 , 
	nIndex:=16#2108 ,   // 平滑时间
	pSrcBuf:=ADR(Par.stDT_date.wSaveCoeCode),      
	cbBufLen:=SIZEOF(Par.stDT_date.wSaveCoeCode),    
	bExecute:= Par.stDT_date.SEPTATLine_SavePara[1],    
	tTimeout:= T#3S, 
	bBusy=> , 
	bError=> , 
	nErrId=> );	
	
//平滑方式参数保存	
FB_EcCoESdoWrite_SEPTATLine[4](
	sNetId:= '192.168.10.10.4.1', 
	nSlaveAddr:=Par.stDT_date.EtherCatAddr[1] ,   //隔膜平移
	nSubIndex:=0 , 
	nIndex:=16#2109 ,   // 平滑方式
	pSrcBuf:=ADR(Par.stDT_date.wSaveCoeCode),      
	cbBufLen:=SIZEOF(Par.stDT_date.wSaveCoeCode),    
	bExecute:= Par.stDT_date.SEPTATLine_SavePara[2],    
	tTimeout:= T#3S, 
	bBusy=> , 
	bError=> , 
	nErrId=> );	

	
//////////////////////////////////////////////////////////////////////一号叠台隔膜缓存
FB_EcCoESdoWrite_SEPTATCache[1](
	sNetId:='192.168.10.10.4.1', 
	nSlaveAddr:=Par.stDT_date.EtherCatAddr[2] ,   //隔膜缓存
	nSubIndex:=0 , 
	nIndex:=16#2108 ,   //  平滑时间
	pSrcBuf:=ADR(Par.stDT_date.SEPTATCache_fSmoothValue[1]),       //写入参数值 
	cbBufLen:=SIZEOF(Par.stDT_date.SEPTATCache_fSmoothValue[1]),    
	bExecute:= Par.stDT_date.SEPTATCache_bWriteCoeValue[1],    
	tTimeout:= T#3S, 
	bBusy=> , 
	bError=> , 
	nErrId=> );
	
FB_EcCoESdoWrite_SEPTATCache[2](
	sNetId:='192.168.10.10.4.1', 
	nSlaveAddr:=Par.stDT_date.EtherCatAddr[2] ,   //隔膜缓存
	nSubIndex:=0 , 
	nIndex:=16#2109 ,   // 平滑方式
	pSrcBuf:=ADR(Par.stDT_date.SEPTATCache_fSmoothValue[2]),       //写入参数值 
	cbBufLen:=SIZEOF(Par.stDT_date.SEPTATCache_fSmoothValue[2]),    
	bExecute:= Par.stDT_date.SEPTATCache_bWriteCoeValue[2],    
	tTimeout:= T#3S, 
	bBusy=> , 
	bError=> , 
	nErrId=> );

//平滑时间参数保存	
FB_EcCoESdoWrite_SEPTATCache[3](
	sNetId:= '192.168.10.10.4.1', 
	nSlaveAddr:=Par.stDT_date.EtherCatAddr[2] ,   //隔膜缓存
	nSubIndex:=0 , 
	nIndex:=16#2108 ,   // 平滑时间
	pSrcBuf:=ADR(Par.stDT_date.wSaveCoeCode),      
	cbBufLen:=SIZEOF(Par.stDT_date.wSaveCoeCode),    
	bExecute:= Par.stDT_date.SEPTATCache_SavePara[1],    
	tTimeout:= T#3S, 
	bBusy=> , 
	bError=> , 
	nErrId=> );	
	
//平滑方式参数保存	
FB_EcCoESdoWrite_SEPTATCache[4](
	sNetId:= '192.168.10.10.4.1', 
	nSlaveAddr:=Par.stDT_date.EtherCatAddr[2] ,   //隔膜缓存
	nSubIndex:=0 , 
	nIndex:=16#2109 ,   // 平滑方式
	pSrcBuf:=ADR(Par.stDT_date.wSaveCoeCode),      
	cbBufLen:=SIZEOF(Par.stDT_date.wSaveCoeCode),    
	bExecute:= Par.stDT_date.SEPTATCache_SavePara[2],    
	tTimeout:= T#3S, 
	bBusy=> , 
	bError=> , 
	nErrId=> );	
	
	
//////////////////////////////////////////////////////////////////////正极送片搬运平移
FB_EcCoESdoWrite_AnCarryingLine[1](
	sNetId:= '192.168.10.10.4.1', 
	nSlaveAddr:=Par.stDT_date.EtherCatAddr[3] ,   //正极送片搬运平移
	nSubIndex:=0 , 
	nIndex:=16#2108 ,   //  平滑时间
	pSrcBuf:=ADR(Par.stDT_date.AnCarryingLine_fSmoothValue[1]),       //写入参数值 
	cbBufLen:=SIZEOF(Par.stDT_date.AnCarryingLine_fSmoothValue[1]),    
	bExecute:= Par.stDT_date.AnCarryingLine_bWriteCoeValue[1],    
	tTimeout:= T#3S, 
	bBusy=> , 
	bError=> , 
	nErrId=> );
	
FB_EcCoESdoWrite_AnCarryingLine[2](
	sNetId:= '192.168.10.10.4.1', 
	nSlaveAddr:=Par.stDT_date.EtherCatAddr[3]  ,   //正极送片搬运平移
	nSubIndex:=0 , 
	nIndex:=16#2109 ,   // 平滑方式
	pSrcBuf:=ADR(Par.stDT_date.AnCarryingLine_fSmoothValue[2]),       //写入参数值 
	cbBufLen:=SIZEOF(Par.stDT_date.AnCarryingLine_fSmoothValue[2]),    
	bExecute:= Par.stDT_date.AnCarryingLine_bWriteCoeValue[2],    
	tTimeout:= T#3S, 
	bBusy=> , 
	bError=> , 
	nErrId=> );

//平滑时间参数保存	
FB_EcCoESdoWrite_AnCarryingLine[3](
	sNetId:= '192.168.10.10.4.1', 
	nSlaveAddr:=Par.stDT_date.EtherCatAddr[3]  ,   //正极送片搬运平移
	nSubIndex:=0 , 
	nIndex:=16#2108 ,   // 平滑时间
	pSrcBuf:=ADR(Par.stDT_date.wSaveCoeCode),      
	cbBufLen:=SIZEOF(Par.stDT_date.wSaveCoeCode),    
	bExecute:= Par.stDT_date.AnCarryingLine_SavePara[1],    
	tTimeout:= T#3S, 
	bBusy=> , 
	bError=> , 
	nErrId=> );	
	
//平滑方式参数保存	
FB_EcCoESdoWrite_AnCarryingLine[4](
	sNetId:= '192.168.10.10.4.1', 
	nSlaveAddr:=Par.stDT_date.EtherCatAddr[3]  ,   //正极送片搬运平移
	nSubIndex:=0 , 
	nIndex:=16#2109 ,   // 平滑方式
	pSrcBuf:=ADR(Par.stDT_date.wSaveCoeCode),      
	cbBufLen:=SIZEOF(Par.stDT_date.wSaveCoeCode),    
	bExecute:= Par.stDT_date.AnCarryingLine_SavePara[2],    
	tTimeout:= T#3S, 
	bBusy=> , 
	bError=> , 
	nErrId=> );		
	
//////////////////////////////////////////////////////////////////////正极叠片搬运平移
FB_EcCoESdoWrite_AnDTCarryingLine[1](
	sNetId:='192.168.10.10.4.1', 
	nSlaveAddr:=Par.stDT_date.EtherCatAddr[4]  ,   //正极叠片搬运平移
	nSubIndex:=0 , 
	nIndex:=16#2108 ,   //  平滑时间
	pSrcBuf:=ADR(Par.stDT_date.AnDTCarryingLine_fSmoothValue[1]),       //写入参数值 
	cbBufLen:=SIZEOF(Par.stDT_date.AnDTCarryingLine_fSmoothValue[1]),    
	bExecute:= Par.stDT_date.AnDTCarryingLine_bWriteCoeValue[1],    
	tTimeout:= T#3S, 
	bBusy=> , 
	bError=> , 
	nErrId=> );
	
FB_EcCoESdoWrite_AnDTCarryingLine[2](
	sNetId:= '192.168.10.10.4.1', 
	nSlaveAddr:=Par.stDT_date.EtherCatAddr[4]  ,   //正极叠片搬运平移
	nSubIndex:=0 , 
	nIndex:=16#2109 ,   // 平滑方式
	pSrcBuf:=ADR(Par.stDT_date.AnDTCarryingLine_fSmoothValue[2]),       //写入参数值 
	cbBufLen:=SIZEOF(Par.stDT_date.AnDTCarryingLine_fSmoothValue[2]),    
	bExecute:= Par.stDT_date.AnDTCarryingLine_bWriteCoeValue[2],    
	tTimeout:= T#3S, 
	bBusy=> , 
	bError=> , 
	nErrId=> );

//平滑时间参数保存	
FB_EcCoESdoWrite_AnDTCarryingLine[3](
	sNetId:= '192.168.10.10.4.1', 
	nSlaveAddr:=Par.stDT_date.EtherCatAddr[4]  ,   //正极叠片搬运平移
	nSubIndex:=0 , 
	nIndex:=16#2108 ,   // 平滑时间
	pSrcBuf:=ADR(Par.stDT_date.wSaveCoeCode),      
	cbBufLen:=SIZEOF(Par.stDT_date.wSaveCoeCode),    
	bExecute:= Par.stDT_date.AnDTCarryingLine_SavePara[1],    
	tTimeout:= T#3S, 
	bBusy=> , 
	bError=> , 
	nErrId=> );	
	
//平滑方式参数保存	
FB_EcCoESdoWrite_AnDTCarryingLine[4](
	sNetId:= '192.168.10.10.4.1', 
	nSlaveAddr:=Par.stDT_date.EtherCatAddr[4]  ,   //正极叠片搬运平移
	nSubIndex:=0 , 
	nIndex:=16#2109 ,   // 平滑方式
	pSrcBuf:=ADR(Par.stDT_date.wSaveCoeCode),      
	cbBufLen:=SIZEOF(Par.stDT_date.wSaveCoeCode),    
	bExecute:= Par.stDT_date.AnDTCarryingLine_SavePara[2],    
	tTimeout:= T#3S, 
	bBusy=> , 
	bError=> , 
	nErrId=> );			
	
//////////////////////////////////////////////////////////////////////负极送片搬运平移
FB_EcCoESdoWrite_CaCarryingLine2[1](
	sNetId:= '192.168.10.10.4.1', 
	nSlaveAddr:=Par.stDT_date.EtherCatAddr[5]  ,   //负极送片搬运平移
	nSubIndex:=0 , 
	nIndex:=16#2108 ,   //  平滑时间
	pSrcBuf:=ADR(Par.stDT_date.CaCarryingLine2_fSmoothValue[1]),       //写入参数值 
	cbBufLen:=SIZEOF(Par.stDT_date.CaCarryingLine2_fSmoothValue[1]),    
	bExecute:= Par.stDT_date.CaCarryingLine2_bWriteCoeValue[1],    
	tTimeout:= T#3S, 
	bBusy=> , 
	bError=> , 
	nErrId=> );
	
FB_EcCoESdoWrite_CaCarryingLine2[2](
	sNetId:= '192.168.10.10.4.1', 
	nSlaveAddr:=Par.stDT_date.EtherCatAddr[5] ,   //负极送片搬运平移
	nSubIndex:=0 , 
	nIndex:=16#2109 ,   // 平滑方式
	pSrcBuf:=ADR(Par.stDT_date.CaCarryingLine2_fSmoothValue[2]),       //写入参数值 
	cbBufLen:=SIZEOF(Par.stDT_date.CaCarryingLine2_fSmoothValue[2]),    
	bExecute:= Par.stDT_date.CaCarryingLine2_bWriteCoeValue[2],    
	tTimeout:= T#3S, 
	bBusy=> , 
	bError=> , 
	nErrId=> );

//平滑时间参数保存	
FB_EcCoESdoWrite_CaCarryingLine2[3](
	sNetId:= '192.168.10.10.4.1', 
	nSlaveAddr:=Par.stDT_date.EtherCatAddr[5] ,   //负极送片搬运平移
	nSubIndex:=0 , 
	nIndex:=16#2108 ,   // 平滑时间
	pSrcBuf:=ADR(Par.stDT_date.wSaveCoeCode),      
	cbBufLen:=SIZEOF(Par.stDT_date.wSaveCoeCode),    
	bExecute:= Par.stDT_date.CaCarryingLine2_SavePara[1],    
	tTimeout:= T#3S, 
	bBusy=> , 
	bError=> , 
	nErrId=> );	
	
//平滑方式参数保存	
FB_EcCoESdoWrite_CaCarryingLine2[4](
	sNetId:='192.168.10.10.4.1', 
	nSlaveAddr:=Par.stDT_date.EtherCatAddr[5] ,   //负极送片搬运平移
	nSubIndex:=0 , 
	nIndex:=16#2109 ,   // 平滑方式
	pSrcBuf:=ADR(Par.stDT_date.wSaveCoeCode),      
	cbBufLen:=SIZEOF(Par.stDT_date.wSaveCoeCode),    
	bExecute:= Par.stDT_date.CaCarryingLine2_SavePara[2],    
	tTimeout:= T#3S, 
	bBusy=> , 
	bError=> , 
	nErrId=> );				
	
//////////////////////////////////////////////////////////////////////负极叠片搬运平移
FB_EcCoESdoWrite_CaDTCarryingLine[1](
	sNetId:= '192.168.10.10.4.1', 
	nSlaveAddr:=Par.stDT_date.EtherCatAddr[6]  ,   //负极叠片搬运平移
	nSubIndex:=0 , 
	nIndex:=16#2108 ,   //  平滑时间
	pSrcBuf:=ADR(Par.stDT_date.CaDTCarryingLine_fSmoothValue[1]),       //写入参数值 
	cbBufLen:=SIZEOF(Par.stDT_date.CaDTCarryingLine_fSmoothValue[1]),    
	bExecute:= Par.stDT_date.CaDTCarryingLine_bWriteCoeValue[1],    
	tTimeout:= T#3S, 
	bBusy=> , 
	bError=> , 
	nErrId=> );
	
FB_EcCoESdoWrite_CaDTCarryingLine[2](
	sNetId:= '192.168.10.10.4.1', 
	nSlaveAddr:=Par.stDT_date.EtherCatAddr[6]  ,   //负极叠片搬运平移
	nSubIndex:=0 , 
	nIndex:=16#2109 ,   // 平滑方式
	pSrcBuf:=ADR(Par.stDT_date.CaDTCarryingLine_fSmoothValue[2]),       //写入参数值 
	cbBufLen:=SIZEOF(Par.stDT_date.CaDTCarryingLine_fSmoothValue[2]),    
	bExecute:= Par.stDT_date.CaDTCarryingLine_bWriteCoeValue[2],    
	tTimeout:= T#3S, 
	bBusy=> , 
	bError=> , 
	nErrId=> );

//平滑时间参数保存	
FB_EcCoESdoWrite_CaDTCarryingLine[3](
	sNetId:= '192.168.10.10.4.1', 
	nSlaveAddr:=Par.stDT_date.EtherCatAddr[6]  ,   //负极叠片搬运平移
	nSubIndex:=0 , 
	nIndex:=16#2108 ,   // 平滑时间
	pSrcBuf:=ADR(Par.stDT_date.wSaveCoeCode),      
	cbBufLen:=SIZEOF(Par.stDT_date.wSaveCoeCode),    
	bExecute:= Par.stDT_date.CaDTCarryingLine_SavePara[1],    
	tTimeout:= T#3S, 
	bBusy=> , 
	bError=> , 
	nErrId=> );	
	
//平滑方式参数保存	
FB_EcCoESdoWrite_CaDTCarryingLine[4](
	sNetId:='192.168.10.10.4.1', 
	nSlaveAddr:=Par.stDT_date.EtherCatAddr[6]  ,   //负极叠片搬运平移
	nSubIndex:=0 , 
	nIndex:=16#2109 ,   // 平滑方式
	pSrcBuf:=ADR(Par.stDT_date.wSaveCoeCode),      
	cbBufLen:=SIZEOF(Par.stDT_date.wSaveCoeCode),    
	bExecute:= Par.stDT_date.CaDTCarryingLine_SavePara[2],    
	tTimeout:= T#3S, 
	bBusy=> , 
	bError=> , 
	nErrId=> );				
	*)
END_ACTION

ACTION P2_Init:
//上电初始化
	CASE Mach_Control.U.Step[0] OF 
			0://等待上电初始化启动
				IF Mach_Control.U.P2Init AND NOT Mach_Control.U.P2InitDone THEN
					Mach_Control.U.Step[0] :=10;
				END_IF
			10://气缸类型初始化,气控阀类型初始化
					//气缸类型初始化
					arrCyCtrl[arrCyNo.CylinderName.	AnScrapbinCy		].Cmd.iType:=	1	;//	正极片NG收纳盒
					arrCyCtrl[arrCyNo.CylinderName.	CaScrapbinCy		].Cmd.iType:=	1	;//	负极片NG收纳盒
					arrCyCtrl[arrCyNo.CylinderName.CaScrapbinUDCy		].Cmd.iType:=	1	;//	负极片NG收纳盒升降
					arrCyCtrl[arrCyNo.CylinderName.	PoleInflationCy		].Cmd.iType:=	3	;//	隔膜放卷气胀轴
					arrCyCtrl[arrCyNo.CylinderName.	PoleTapeSplicerLCy		].Cmd.iType:=	1	;//	隔膜接带左压板气缸
					arrCyCtrl[arrCyNo.CylinderName.	PoleTapeSplicerRCy		].Cmd.iType:=	1	;//	隔膜接带右压板气缸
					arrCyCtrl[arrCyNo.CylinderName.PreDiaph		].Cmd.iType:=	1	;//	叠台压隔膜气缸
					arrCyCtrl[arrCyNo.CylinderName.	PoleTapeCy		].Cmd.iType:=	1	;//	隔膜夹紧气缸
					arrCyCtrl[arrCyNo.CylinderName.	PoleHotCutterCy		].Cmd.iType:=	1	;//	隔膜热切升降
					arrCyCtrl[arrCyNo.CylinderName.	PoleSplintCy_U		].Cmd.iType:=	1	;//	夹膜上夹板
					arrCyCtrl[arrCyNo.CylinderName.	PoleSplintCy_D		].Cmd.iType:=	1	;//	夹膜下夹板
					arrCyCtrl[arrCyNo.CylinderName.	TailCurlSplintCy		].Cmd.iType:=	1	;//	尾卷夹爪开合
					arrCyCtrl[arrCyNo.CylinderName.	CurlingSplintCy_L		].Cmd.iType:=	3	;//	长卷针夹开合
					arrCyCtrl[arrCyNo.CylinderName.	CurlingSplintCy_S		].Cmd.iType:=	3	;//	短卷针夹开合
					//arrCyCtrl[arrCyNo.CylinderName.	CurlingSplintCy_S_1		].Cmd.iType:=	2	;//	短卷针夹开合_1
					arrCyCtrl[arrCyNo.CylinderName.	TailCurlLineCy		].Cmd.iType:=	1	;//	尾卷压辊平移缸
					arrCyCtrl[arrCyNo.CylinderName.	TailCurlUpdownCy		].Cmd.iType:=	1	;//	尾卷压辊升降缸
					arrCyCtrl[arrCyNo.CylinderName.	StandbyGlueCy		].Cmd.iType:=	2	;//	备胶气缸
					arrCyCtrl[arrCyNo.CylinderName.	CodeStandbyGlueCy		].Cmd.iType:=	2	;//	备二维码胶气缸
					arrCyCtrl[arrCyNo.CylinderName.	GlueClampsCy		].Cmd.iType:=	1	;//	贴胶夹爪气缸
					arrCyCtrl[arrCyNo.CylinderName.	GluePressCy		].Cmd.iType:=	1	;//	压胶气缸
					arrCyCtrl[arrCyNo.CylinderName.	CodeGluePressCy		].Cmd.iType:=	1	;//	压二维码胶气缸
					arrCyCtrl[arrCyNo.CylinderName.	GlueCutCy		].Cmd.iType:=	1	;//	切胶气缸
					arrCyCtrl[arrCyNo.CylinderName.	codeGlueCutCy		].Cmd.iType:=	1	;//	切二维码胶气缸
					arrCyCtrl[arrCyNo.CylinderName.	PullGluePoleCy		].Cmd.iType:=	4	;//	拉胶杆抱紧
					arrCyCtrl[arrCyNo.CylinderName.	PullGlueCy		].Cmd.iType:=	1	;//	拉胶气缸
					arrCyCtrl[arrCyNo.CylinderName.	GlueNGCy		].Cmd.iType:=	1	;//	踢废胶气缸
					arrCyCtrl[arrCyNo.CylinderName.	PullGlueModelCy		].Cmd.iType:=	1	;//	贴胶治具气缸
					//气控阀类型初始化				
					arrCyCtrl[arrCyNo.ElectValveName.	AnBeltVacuum		].Cmd.iType:=	4	;//	正极模切送料分段皮带1取料处真空
					arrCyCtrl[arrCyNo.ElectValveName.	AnBeltVacuumBark		].Cmd.iType:=	4	;//	正极模切送料分段皮带1取料处破真空
					arrCyCtrl[arrCyNo.ElectValveName.	CaMQBeltVacuum		].Cmd.iType:=	4	;//	负极模切送料分段皮带1取料处真空
					arrCyCtrl[arrCyNo.ElectValveName.	CaMQBeltVacuumBark		].Cmd.iType:=	4	;//	负极模切送料分段皮带1取料处破真空
					arrCyCtrl[arrCyNo.ElectValveName.	AnCarryingVacuum		].Cmd.iType:=	4	;//	正极送片搬运升降真空
					arrCyCtrl[arrCyNo.ElectValveName.	AnCarryingVacuumBark		].Cmd.iType:=	4	;//	正极送片搬运升降破真空
					arrCyCtrl[arrCyNo.ElectValveName.	AndeviationVacuum		].Cmd.iType:=	4	;//	正极纠偏平台真空
					arrCyCtrl[arrCyNo.ElectValveName.	AndeviationIonizedWind		].Cmd.iType:=	4	;//	正极纠偏平台除尘风刀
					arrCyCtrl[arrCyNo.ElectValveName.	AndeviationVacuumBark		].Cmd.iType:=	4	;//	正极纠偏平台破真空
					arrCyCtrl[arrCyNo.ElectValveName.	AnDTCarryingVacuum		].Cmd.iType:=	4	;//	正极叠片搬运升降真空
					//arrCyCtrl[arrCyNo.ElectValveName.	AnDTCarryingJRVacuum		].Cmd.iType:=	4	;//	正极叠台搬运升降极耳真空
					arrCyCtrl[arrCyNo.ElectValveName.	AnDTCarryingVacuumBark		].Cmd.iType:=	4	;//	正极叠片搬运升降破真空
					arrCyCtrl[arrCyNo.ElectValveName.	CaCarryingVacuum1		].Cmd.iType:=	4	;//	负极送片搬运升降1真空
					arrCyCtrl[arrCyNo.ElectValveName.	CaCarryingVacuumBark1		].Cmd.iType:=	4	;//	负极送片搬运升降1破真空
					arrCyCtrl[arrCyNo.ElectValveName.	CaLoadUpBeltVacuum		].Cmd.iType:=	4	;//	负极送片皮带末端真空
					arrCyCtrl[arrCyNo.ElectValveName.	CaLoadUpBeltVacuumBark		].Cmd.iType:=	4	;//	负极送片皮带末端破真空
					arrCyCtrl[arrCyNo.ElectValveName.	CaCarryingVacuum2		].Cmd.iType:=	4	;//	负极送片搬运升降2真空
					arrCyCtrl[arrCyNo.ElectValveName.	CaCarryingVacuumBark2		].Cmd.iType:=	4	;//	负极送片搬运升降2破真空
					arrCyCtrl[arrCyNo.ElectValveName.	CadeviationVacuum		].Cmd.iType:=	4	;//	负极纠偏平台真空
					arrCyCtrl[arrCyNo.ElectValveName.	CadeviationVacuumBark		].Cmd.iType:=	4	;//	负极纠偏平台破真空
					arrCyCtrl[arrCyNo.ElectValveName.	CadeviationIonizedWind		].Cmd.iType:=	4	;//	负极纠偏平台除尘风刀
					arrCyCtrl[arrCyNo.ElectValveName.	CaDTCarryingVacuum		].Cmd.iType:=	4	;//	负极叠片搬运升降真空
					//arrCyCtrl[arrCyNo.ElectValveName.	CaDTCarryingJRVacuum		].Cmd.iType:=	4	;//	负极叠片搬运升降极耳真空
					arrCyCtrl[arrCyNo.ElectValveName.	CaDTCarryingVacuumBark		].Cmd.iType:=	4	;//	负极叠片搬运升降破真空
					arrCyCtrl[arrCyNo.ElectValveName.	PoleTapeDustRemoval		].Cmd.iType:=	4	;//	隔膜接带平台除尘
					arrCyCtrl[arrCyNo.ElectValveName.	PoleTapeVacuum		].Cmd.iType:=	4	;//	隔膜接带平台真空
					arrCyCtrl[arrCyNo.ElectValveName.	BlueGlueVacuum1		].Cmd.iType:=	4	;//	备胶组件蓝胶真空1
					arrCyCtrl[arrCyNo.ElectValveName.	BlueGlueVacuum2		].Cmd.iType:=	4	;//	备胶组件蓝胶真空2
					arrCyCtrl[arrCyNo.ElectValveName.	codeGlueVacuum1		].Cmd.iType:=	4	;//	备胶组件二维码胶真空1
					arrCyCtrl[arrCyNo.ElectValveName.	codeGlueVacuum2		].Cmd.iType:=	4	;//	备胶组件二维码胶真空2
					arrCyCtrl[arrCyNo.ElectValveName.	PastesGlueVacuum		].Cmd.iType:=	4	;//	备胶组件贴胶头真空
					arrCyCtrl[arrCyNo.ElectValveName.	DTVacuum		].Cmd.iType:=	4	;//	叠片台真空
					arrCyCtrl[arrCyNo.ElectValveName.	PoleSplintVacuum_D		].Cmd.iType:=	4	;//	夹膜下夹板真空
					arrCyCtrl[arrCyNo.ElectValveName.WJ_blow		].Cmd.iType:=	4	;//	夹电芯吹气
					arrCyCtrl[arrCyNo.ElectValveName.WJShortvacuum		].Cmd.iType:=	4	;//短卷针张开真空
					//屏蔽初赋值					
					Mach_Control.U.Step[0] :=20;
					
			20://计算从左到右、从右到左移动时隔膜变化量
					CaCrectCamStep0:=10;//负极取片凸轮创建
					AnCrectCamStep0:=10;//正极取片凸轮创建
					YDCrectCamStep0:=10;//叠台压刀凸轮创建
					GMCreatCamStep0:=10;//叠台缓存凸轮创建
					WZCreatCamStep0:=10;//尾卷凸轮创建
					Mach_Control.U.Step[0] :=30;
			30://判断隔膜变数据是否完成
					IF CaCrectCamStep0=6666 AND AnCrectCamStep0=6666 AND YDCrectCamStep0=6666 AND  GMCreatCamStep0=6666 AND WZCreatCamStep0=6666 THEN
						Mach_Control.U.Step[0] :=40;
					END_IF;
			40:
				arrCyCtrl[arrCyNo.CylinderName.PoleInflationCy].Cmd.bON:=TRUE;
				Mach_Control.U.P2Init :=FALSE;//复位上电初始化完成
				Mach_Control.U.P2InitDone:=TRUE;//置位上电初始化完成
				Mach_Control.U.Step[0] :=0;
	END_CASE

	arrCyCtrl[arrCyNo.ElectValveName.	CaCarryingVacuumBark2		].Cmd.bON;
END_ACTION

ACTION Stick_Condition:
//贴胶平移，贴胶旋转轴移动允许  AND  arrAxisCtrl[AxiseNo.AxisName.TailCurlLine].Status.fSetPos>=arrAxisPar[AxiseNo.AxisName.TailCurlLine].arrTargetPoint[1]+0.2 AND arrAxisPar[AxiseNo.AxisName.TailCurlWhirling].arrTargetPoint[1] 
IF arrAxisCtrl[AxiseNo.AxisName.GluingRetracting].Status.Homed 
AND arrAxisCtrl[AxiseNo.AxisName.GluingRetracting].Status.NoMoving 
AND arrAxisCtrl[AxiseNo.AxisName.GluingRetracting].Cmd.arrbRealPoint[1] 
AND  ((arrAxisCtrl[AxiseNo.AxisName.TailCurlLine].Status.fSetPos>=arrAxisPar[AxiseNo.AxisName.TailCurlLine].arrTargetPoint[1]-1 AND  arrAxisCtrl[AxiseNo.AxisName.TailCurlRetracting].Status.fSetPos<=arrAxisPar[AxiseNo.AxisName.TailCurlRetracting].arrTargetPoint[1]+1) OR
		 arrAxisCtrl[AxiseNo.AxisName.TailCurlWhirling].Cmd.arrbRealPoint[1]  )
AND  ((DTselect=1 AND (arrAxisCtrl[P3AxisNo.P3M1_ColdpreLine].Status.fActPos <=  arrAxisPar[P3AxisNo.P3M1_ColdpreLine].arrTargetPoint[2]-300 OR 
            arrAxisCtrl[P3AxisNo.P3M1_ColdpreLine].Status.fActPos >=  arrAxisPar[P3AxisNo.P3M1_ColdpreLine].arrTargetPoint[2]+300)) OR    
         (DTselect=2 AND (arrAxisCtrl[P3AxisNo.P3M1_ColdpreLine].Status.fActPos <=  arrAxisPar[P3AxisNo.P3M1_ColdpreLine].arrTargetPoint[3]-300 OR 
			 arrAxisCtrl[P3AxisNo.P3M1_ColdpreLine].Status.fActPos >=  arrAxisPar[P3AxisNo.P3M1_ColdpreLine].arrTargetPoint[3]+300)) OR
		 (DTselect=3 AND (arrAxisCtrl[P3AxisNo.P3M1_ColdpreLine].Status.fActPos <=  arrAxisPar[P3AxisNo.P3M1_ColdpreLine].arrTargetPoint[4]-300 OR 
			 arrAxisCtrl[P3AxisNo.P3M1_ColdpreLine].Status.fActPos >=  arrAxisPar[P3AxisNo.P3M1_ColdpreLine].arrTargetPoint[4]+300))  OR 
		( arrAxisCtrl[P3AxisNo.P3M1_ColdpreWhirling].Cmd.arrbRealPoint[1] OR arrAxisCtrl[P3AxisNo.P3M1_ColdpreWhirling].Cmd.arrbRealPoint[5] OR arrAxisCtrl[P3AxisNo.P3M1_ColdpreWhirling].Cmd.arrbRealPoint[6]) )
(*AND arrAxisCtrl[AxiseNo.AxisName.TailCurlLine].Status.Homed 
AND  arrAxisCtrl[AxiseNo.AxisName.TailCurlRetracting].Cmd.arrbRealPoint[1] 
AND arrAxisCtrl[AxiseNo.AxisName.TailCurlRetracting].Status.Homed 
AND(((arrAxisCtrl[AxiseNo.AxisName.TailCurlLine].Status.fSetPos>= (arrAxisPar[AxiseNo.AxisName.TailCurlLine].arrTargetPoint[1]-1) 
AND (arrAxisCtrl[AxiseNo.AxisName.TailCurlWhirling].Cmd.arrbRealPoint[1] 
OR arrAxisCtrl[AxiseNo.AxisName.TailCurlWhirling].Cmd.arrbRealPoint[3] 
OR  arrAxisCtrl[AxiseNo.AxisName.TailCurlWhirling].Cmd.arrbRealPoint[4])) 
OR((arrAxisCtrl[AxiseNo.AxisName.TailCurlLine].Status.fSetPos>= (arrAxisPar[AxiseNo.AxisName.TailCurlLine].arrTargetPoint[5]-1)) 
AND arrAxisCtrl[AxiseNo.AxisName.TailCurlWhirling].Cmd.arrbRealPoint[2])))*)    THEN
	arrAxisCtrl[AxiseNo.AxisName.GluingLine].Cmd.GoPoint_Condition[0]:=TRUE;
	GluingLineagree:=TRUE;//侧贴胶平移轴、侧贴胶旋转轴动作允许
ELSE
	GluingLineagree:=FALSE;
	arrAxisCtrl[AxiseNo.AxisName.GluingLine].Cmd.GoPoint_Condition[0]:=FALSE;
END_IF


//贴胶旋转轴移动允许
IF GluingLineagree THEN
	GluingWhirlingagree:=TRUE;//侧贴胶平移轴、侧贴胶旋转轴动作允许
ELSE
	GluingWhirlingagree:=FALSE;
END_IF


Mach_Control.TJ_b.WhirlingSafe:=(*arrAxisCtrl[AxiseNo.AxisName.GluingWhirling].Status.Homed AND arrAxisCtrl[AxiseNo.AxisName.GluingWhirling].Status.NoMoving
                        AND*) arrAxisCtrl[AxiseNo.AxisName.GluingRetracting].Status.Homed AND arrAxisCtrl[AxiseNo.AxisName.GluingRetracting].Cmd.arrbRealPoint[1]
						AND (arrAxisCtrl[AxiseNo.AxisName.GluingLine].Status.fActPos <= (arrAxisPar[AxiseNo.AxisName.GluingLine].arrTargetPoint[10]+1)) AND
                         ((DTselect=1 AND (arrAxisCtrl[P3AxisNo.P3M1_ColdpreLine].Status.fActPos <=  arrAxisPar[P3AxisNo.P3M1_ColdpreLine].arrTargetPoint[2]-300 OR 
                              arrAxisCtrl[P3AxisNo.P3M1_ColdpreLine].Status.fActPos >=  arrAxisPar[P3AxisNo.P3M1_ColdpreLine].arrTargetPoint[2]+300)) OR
						(DTselect=2 AND (arrAxisCtrl[P3AxisNo.P3M1_ColdpreLine].Status.fActPos <=  arrAxisPar[P3AxisNo.P3M1_ColdpreLine].arrTargetPoint[3]-300 OR 
													  arrAxisCtrl[P3AxisNo.P3M1_ColdpreLine].Status.fActPos >=  arrAxisPar[P3AxisNo.P3M1_ColdpreLine].arrTargetPoint[3]+300)) OR
						(DTselect=3 AND (arrAxisCtrl[P3AxisNo.P3M1_ColdpreLine].Status.fActPos <=  arrAxisPar[P3AxisNo.P3M1_ColdpreLine].arrTargetPoint[4]-300 OR 
													  arrAxisCtrl[P3AxisNo.P3M1_ColdpreLine].Status.fActPos >=  arrAxisPar[P3AxisNo.P3M1_ColdpreLine].arrTargetPoint[4]+300))  OR 
						 ( arrAxisCtrl[P3AxisNo.P3M1_ColdpreWhirling].Cmd.arrbRealPoint[1] OR arrAxisCtrl[P3AxisNo.P3M1_ColdpreWhirling].Cmd.arrbRealPoint[5] OR arrAxisCtrl[P3AxisNo.P3M1_ColdpreWhirling].Cmd.arrbRealPoint[6]) );

					//AND (arrAxisCtrl[AxiseNo.AxisName.GluingLine].Status.fSetPos >= (arrAxisPar[AxiseNo.AxisName.GluingLine].arrTargetPoint[10]-1));

//侧贴胶平移运动允许
arrAxisCtrl[AxiseNo.AxisName.GluingLine].Cmd.GoPoint_Condition[0]:=GluingLineagree OR Mach_Control.TJ_b.AxisConditionEN ;
arrAxisCtrl[AxiseNo.AxisName.GluingLine].Cmd.GoPoint_Condition[1]:=GluingLineagree OR Mach_Control.TJ_b.AxisConditionEN ;
//侧贴胶旋转运动允许
arrAxisCtrl[AxiseNo.AxisName.GluingWhirling].Cmd.GoPoint_Condition[0]:=GluingLineagree OR Mach_Control.TJ_b.AxisConditionEN ;
arrAxisCtrl[AxiseNo.AxisName.GluingWhirling].Cmd.GoPoint_Condition[1]:=GluingLineagree OR Mach_Control.TJ_b.AxisConditionEN ;


//侧贴胶平移、旋转在下料位，侧贴胶夹爪气缸张开，允许尾卷下电芯
IF arrAxisCtrl[AxiseNo.AxisName.GluingLine].Status.Homed AND arrAxisCtrl[AxiseNo.AxisName.GluingLine].Status.NoMoving AND arrAxisCtrl[AxiseNo.AxisName.GluingLine].Cmd.arrbRealPoint[1] AND 
	 arrAxisCtrl[AxiseNo.AxisName.GluingWhirling].Status.Homed AND arrAxisCtrl[AxiseNo.AxisName.GluingWhirling].Status.NoMoving AND arrAxisCtrl[AxiseNo.AxisName.GluingWhirling].Cmd.arrbRealPoint[1] AND
	arrCyCtrl[arrCyNo.CylinderName.GlueClampsCy].Io.DIOnSwitch THEN
	Mach_Control.TJ_b.Stickerragree:=TRUE;	
ELSE
	Mach_Control.TJ_b.Stickerragree:=FALSE;		
END_IF
//贴胶完成，允许冷压取电芯
IF Mach_Control.TJ_b.StickerDone AND Mach_Control.TJ_b.StickerFlag AND arrAxisCtrl[AxiseNo.AxisName.GluingLine].Cmd.arrbRealPoint[2] AND arrAxisCtrl[AxiseNo.AxisName.GluingWhirling].Cmd.arrbRealPoint[2]  THEN
	Mach_Control.TJ_b.StickerOffloading:=TRUE;
ELSE
	Mach_Control.TJ_b.StickerOffloading:=FALSE; 	
END_IF
//拉胶在安全位，允许贴胶头前进、后退
IF arrAxisCtrl[AxiseNo.AxisName.GluingUpDown].Status.Homed AND arrAxisCtrl[AxiseNo.AxisName.GluingUpDown].Status.NoMoving AND 
	(arrAxisCtrl[AxiseNo.AxisName.GluingUpDown].Status.fActPos<= arrAxisPar[AxiseNo.AxisName.GluingUpDown].arrTargetPoint[4] OR
	arrAxisCtrl[AxiseNo.AxisName.GluingUpDown].Status.fActPos>= arrAxisPar[AxiseNo.AxisName.GluingUpDown].arrTargetPoint[2]) 
	AND arrCyCtrl[arrCyNo.CylinderName.GlueClampsCy].Status.OFFState THEN
	GluingRetractingagree:=TRUE;//贴胶头前进轴动作允许
ELSE
	GluingRetractingagree:=FALSE;
END_IF

arrAxisCtrl[AxiseNo.AxisName.GluingRetracting].Cmd.GoPoint_Condition[0]:=GluingRetractingagree OR Mach_Control.TJ_b.AxisConditionEN ;
arrAxisCtrl[AxiseNo.AxisName.GluingRetracting].Cmd.GoPoint_Condition[1]:=GluingRetractingagree OR Mach_Control.TJ_b.AxisConditionEN ;
arrAxisCtrl[AxiseNo.AxisName.GluingRetracting].Cmd.GoPoint_Condition[2]:=GluingRetractingagree OR Mach_Control.TJ_b.AxisConditionEN ;
arrAxisCtrl[AxiseNo.AxisName.GluingRetracting].Cmd.GoPoint_Condition[3]:=GluingRetractingagree OR Mach_Control.TJ_b.AxisConditionEN ;
arrAxisCtrl[AxiseNo.AxisName.GluingRetracting].Cmd.GoPoint_Condition[4]:=GluingRetractingagree OR Mach_Control.TJ_b.AxisConditionEN ;
arrAxisCtrl[AxiseNo.AxisName.GluingRetracting].Cmd.GoPoint_Condition[5]:=GluingRetractingagree OR Mach_Control.TJ_b.AxisConditionEN ;
//拉胶升降允许动作
IF arrAxisCtrl[AxiseNo.AxisName.GluingRetracting].Status.Homed AND 
	arrAxisCtrl[AxiseNo.AxisName.GluingRetracting].Status.fActPos<= arrAxisPar[AxiseNo.AxisName.GluingRetracting].arrTargetPoint[1]+0.2 AND 
	arrCyCtrl[arrCyNo.CylinderName.codeGlueCutCy].Status.ONState AND
	arrCyCtrl[arrCyNo.CylinderName.GlueCutCy].Status.ONState AND
	arrCyCtrl[arrCyNo.CylinderName.GlueNGCy].Status.OFFState AND 
	arrCyCtrl[arrCyNo.CylinderName.PullGlueCy].Status.ONState  THEN
	GluingUpDownagree:=TRUE; 
ELSE
	GluingUpDownagree:=false;	
END_IF
arrAxisCtrl[AxiseNo.AxisName.GluingUpDown].Cmd.GoPoint_Condition[1]:=GluingUpDownagree OR Mach_Control.TJ_b.AxisConditionEN ;	
arrAxisCtrl[AxiseNo.AxisName.GluingUpDown].Cmd.GoPoint_Condition[2]:=GluingUpDownagree OR Mach_Control.TJ_b.AxisConditionEN ;	
arrAxisCtrl[AxiseNo.AxisName.GluingUpDown].Cmd.GoPoint_Condition[3]:=GluingUpDownagree OR Mach_Control.TJ_b.AxisConditionEN ;	
arrAxisCtrl[AxiseNo.AxisName.GluingUpDown].Cmd.GoPoint_Condition[4]:=GluingUpDownagree OR Mach_Control.TJ_b.AxisConditionEN ;	
arrAxisCtrl[AxiseNo.AxisName.GluingUpDown].Cmd.GoPoint_Condition[5]:=GluingUpDownagree OR Mach_Control.TJ_b.AxisConditionEN ;	
arrAxisCtrl[AxiseNo.AxisName.GluingUpDown].Cmd.GoPoint_Condition[6]:=GluingUpDownagree OR Mach_Control.TJ_b.AxisConditionEN ;	
arrAxisCtrl[AxiseNo.AxisName.GluingUpDown].Cmd.GoPoint_Condition[7]:=GluingUpDownagree OR Mach_Control.TJ_b.AxisConditionEN ;	
arrAxisCtrl[AxiseNo.AxisName.GluingUpDown].Cmd.GoPoint_Condition[8]:=GluingUpDownagree OR Mach_Control.TJ_b.AxisConditionEN ;	


//气缸条件
IF arrCyCtrl[arrCyNo.CylinderName.GlueCutCy].Status.OFFState AND arrCyCtrl[arrCyNo.CylinderName.GlueCutCy].Status.OFFState  THEN
	arrCyCtrl[arrCyNo.CylinderName.GlueNGCy].Cmd.OnCondition:=TRUE;
ELSE
	arrCyCtrl[arrCyNo.CylinderName.GlueNGCy].Cmd.OnCondition:=FALSE;
END_IF

/////////////////////////////////////////////////////////////
/////////////////////////////////////////////////////////
////////////////////////////////////////////电机条件
//侧贴胶平移
IF  Mach_Control.U.WJ_iMode=3 
  AND GluingLineagree
 OR Mach_Control.TJ_b.AxisConditionEN THEN
	arrAxisCtrl[AxiseNo.AxisName.GluingLine].Cmd.Home_Condition:=TRUE;
ELSE
	arrAxisCtrl[AxiseNo.AxisName.GluingLine].Cmd.Home_Condition:=FALSE;	
END_IF

IF  Mach_Control.U.WJ_iMode=3 
AND arrAxisCtrl[AxiseNo.AxisName.GluingLine].Status.Homed 
AND GluingLineagree
 OR Mach_Control.TJ_b.AxisConditionEN THEN
	arrAxisCtrl[AxiseNo.AxisName.GluingLine].Cmd.GoPoint_Condition[1]:=TRUE;
ELSE
	arrAxisCtrl[AxiseNo.AxisName.GluingLine].Cmd.GoPoint_Condition[1]:=FALSE;	
END_IF

IF  Mach_Control.U.WJ_iMode=3 
AND arrAxisCtrl[AxiseNo.AxisName.GluingLine].Status.Homed 
AND GluingLineagree
 OR Mach_Control.TJ_b.AxisConditionEN THEN
	arrAxisCtrl[AxiseNo.AxisName.GluingLine].Cmd.GoPoint_Condition[2]:=TRUE;
ELSE
	arrAxisCtrl[AxiseNo.AxisName.GluingLine].Cmd.GoPoint_Condition[2]:=FALSE;	
END_IF

IF  Mach_Control.U.WJ_iMode=3 
AND arrAxisCtrl[AxiseNo.AxisName.GluingLine].Status.Homed 
AND GluingLineagree
 OR Mach_Control.TJ_b.AxisConditionEN THEN
	arrAxisCtrl[AxiseNo.AxisName.GluingLine].Cmd.GoPoint_Condition[3]:=TRUE;
ELSE
	arrAxisCtrl[AxiseNo.AxisName.GluingLine].Cmd.GoPoint_Condition[3]:=FALSE;	
END_IF

IF  Mach_Control.U.WJ_iMode=3 
AND arrAxisCtrl[AxiseNo.AxisName.GluingLine].Status.Homed 
AND GluingLineagree
 OR Mach_Control.TJ_b.AxisConditionEN THEN
	arrAxisCtrl[AxiseNo.AxisName.GluingLine].Cmd.GoPoint_Condition[4]:=TRUE;
ELSE
	arrAxisCtrl[AxiseNo.AxisName.GluingLine].Cmd.GoPoint_Condition[4]:=FALSE;	
END_IF

IF  Mach_Control.U.WJ_iMode=3 
AND arrAxisCtrl[AxiseNo.AxisName.GluingLine].Status.Homed  
AND GluingLineagree
 OR Mach_Control.TJ_b.AxisConditionEN THEN
	arrAxisCtrl[AxiseNo.AxisName.GluingLine].Cmd.GoPoint_Condition[5]:=TRUE;
ELSE
	arrAxisCtrl[AxiseNo.AxisName.GluingLine].Cmd.GoPoint_Condition[5]:=FALSE;	
END_IF

IF  Mach_Control.U.WJ_iMode=3 
AND arrAxisCtrl[AxiseNo.AxisName.GluingLine].Status.Homed  
AND GluingLineagree
 OR Mach_Control.TJ_b.AxisConditionEN THEN
	arrAxisCtrl[AxiseNo.AxisName.GluingLine].Cmd.GoPoint_Condition[6]:=TRUE;
ELSE
	arrAxisCtrl[AxiseNo.AxisName.GluingLine].Cmd.GoPoint_Condition[6]:=FALSE;	
END_IF

IF  Mach_Control.U.WJ_iMode=3 
AND arrAxisCtrl[AxiseNo.AxisName.GluingLine].Status.Homed 
AND GluingLineagree
OR Mach_Control.TJ_b.AxisConditionEN THEN
	arrAxisCtrl[AxiseNo.AxisName.GluingLine].Cmd.GoPoint_Condition[8]:=TRUE;
ELSE
	arrAxisCtrl[AxiseNo.AxisName.GluingLine].Cmd.GoPoint_Condition[8]:=FALSE;	
END_IF

IF  Mach_Control.U.WJ_iMode=3 
AND arrAxisCtrl[AxiseNo.AxisName.GluingLine].Status.Homed 
AND GluingLineagree
OR Mach_Control.TJ_b.AxisConditionEN  THEN
	arrAxisCtrl[AxiseNo.AxisName.GluingLine].Cmd.GoPoint_Condition[9]:=TRUE;
ELSE
	arrAxisCtrl[AxiseNo.AxisName.GluingLine].Cmd.GoPoint_Condition[9]:=FALSE;	
END_IF

IF  Mach_Control.U.WJ_iMode=3 
AND arrAxisCtrl[AxiseNo.AxisName.GluingLine].Status.Homed 
AND GluingLineagree
 OR Mach_Control.TJ_b.AxisConditionEN THEN
	arrAxisCtrl[AxiseNo.AxisName.GluingLine].Cmd.GoPoint_Condition[10]:=TRUE;
ELSE
	arrAxisCtrl[AxiseNo.AxisName.GluingLine].Cmd.GoPoint_Condition[10]:=FALSE;	
END_IF

//侧贴胶旋转//暂时屏蔽冷压
IF  Mach_Control.U.WJ_iMode=3 
//AND arrAxisCtrl[AxiseNo.AxisName.GluingWhirling].Status.Homed  
AND Mach_Control.TJ_b.WhirlingSafe
OR Mach_Control.TJ_b.AxisConditionEN THEN
	arrAxisCtrl[AxiseNo.AxisName.GluingWhirling].Cmd.Home_Condition:=TRUE;
ELSE
	arrAxisCtrl[AxiseNo.AxisName.GluingWhirling].Cmd.Home_Condition:=FALSE;	
END_IF

IF  Mach_Control.U.WJ_iMode=3 
AND arrAxisCtrl[AxiseNo.AxisName.GluingWhirling].Status.Homed  
AND arrAxisCtrl[AxiseNo.AxisName.GluingRetracting].Cmd.arrbRealPoint[1] 
AND ((arrAxisCtrl[AxiseNo.AxisName.TailCurlLine].Status.fSetPos>=arrAxisPar[AxiseNo.AxisName.TailCurlLine].arrTargetPoint[10]-1 
AND  arrAxisCtrl[AxiseNo.AxisName.TailCurlRetracting].Status.fSetPos<=arrAxisPar[AxiseNo.AxisName.TailCurlRetracting].arrTargetPoint[1]+1) OR arrAxisCtrl[AxiseNo.AxisName.TailCurlWhirling].Cmd.arrbRealPoint[1]) 
AND ((arrAxisCtrl[P3AxisNo.P3M1_ColdpreWhirling].Cmd.arrbRealPoint[1] 
OR arrAxisCtrl[P3AxisNo.P3M1_ColdpreWhirling].Cmd.arrbRealPoint[5]
OR arrAxisCtrl[P3AxisNo.P3M1_ColdpreWhirling].Cmd.arrbRealPoint[6] ) 
(*OR arrAxisCtrl[P3AxisNo.P3M1_ColdpreRetracting].Cmd.arrbRealPoint[1]*))
AND NOT arrAxisCtrl[AxiseNo.AxisName.GluingLine].Cmd.arrbRealPoint[8]
OR Mach_Control.TJ_b.AxisConditionEN THEN
	arrAxisCtrl[AxiseNo.AxisName.GluingWhirling].Cmd.GoPoint_Condition[1]:=TRUE;
	arrAxisCtrl[AxiseNo.AxisName.GluingWhirling].Cmd.GoPoint_Condition[2]:=TRUE;
	arrAxisCtrl[AxiseNo.AxisName.GluingWhirling].Cmd.GoPoint_Condition[3]:=TRUE;
	arrAxisCtrl[AxiseNo.AxisName.GluingWhirling].Cmd.GoPoint_Condition[4]:=TRUE;
	arrAxisCtrl[AxiseNo.AxisName.GluingWhirling].Cmd.GoPoint_Condition[5]:=TRUE;
	arrAxisCtrl[AxiseNo.AxisName.GluingWhirling].Cmd.GoPoint_Condition[6]:=TRUE;
ELSE
	arrAxisCtrl[AxiseNo.AxisName.GluingWhirling].Cmd.GoPoint_Condition[1]:=FALSE;
	arrAxisCtrl[AxiseNo.AxisName.GluingWhirling].Cmd.GoPoint_Condition[2]:=FALSE;
	arrAxisCtrl[AxiseNo.AxisName.GluingWhirling].Cmd.GoPoint_Condition[3]:=FALSE;
	arrAxisCtrl[AxiseNo.AxisName.GluingWhirling].Cmd.GoPoint_Condition[4]:=TRUE;
	arrAxisCtrl[AxiseNo.AxisName.GluingWhirling].Cmd.GoPoint_Condition[5]:=FALSE;
	arrAxisCtrl[AxiseNo.AxisName.GluingWhirling].Cmd.GoPoint_Condition[6]:=FALSE;	
END_IF
(*
IF  Mach_Control.U.WJ_iMode=3 AND arrAxisCtrl[AxiseNo.AxisName.GluingWhirling].Status.Homed  AND arrAxisCtrl[AxiseNo.AxisName.GluingRetracting].Cmd.arrbRealPoint[1] 
AND  ((arrAxisCtrl[AxiseNo.AxisName.TailCurlLine].Status.fSetPos>=arrAxisPar[AxiseNo.AxisName.TailCurlLine].arrTargetPoint[1]-1 AND  arrAxisCtrl[AxiseNo.AxisName.TailCurlRetracting].Status.fSetPos<=arrAxisPar[AxiseNo.AxisName.TailCurlRetracting].arrTargetPoint[1]+1) OR
    	  arrAxisCtrl[AxiseNo.AxisName.TailCurlWhirling].Cmd.arrbRealPoint[1]  ) 
 AND  ( (  arrAxisCtrl[P3AxisNo.P3M1_ColdpreWhirling].Cmd.arrbRealPoint[1] OR arrAxisCtrl[P3AxisNo.P3M1_ColdpreWhirling].Cmd.arrbRealPoint[5] OR arrAxisCtrl[P3AxisNo.P3M1_ColdpreWhirling].Cmd.arrbRealPoint[6] ) OR
                    arrAxisCtrl[P3AxisNo.P3M1_ColdpreRetracting].Cmd.arrbRealPoint[1] )
 OR Mach_Control.TJ_b.AxisConditionEN THEN
	arrAxisCtrl[AxiseNo.AxisName.GluingWhirling].Cmd.GoPoint_Condition[2]:=TRUE;
ELSE
	arrAxisCtrl[AxiseNo.AxisName.GluingWhirling].Cmd.GoPoint_Condition[2]:=FALSE;	
END_IF

